{attribute 'monitoring' := 'call'}
PROPERTY PRIVATE HomeSpeedZ : LREAL
GET
HomeSpeedZ := stLocalSettings.stDynStationSettings[E_St030_Settings.eSt030_Settings_ZHomeSpeed].fValue;
END_GET
END_PROPERTY

{attribute 'monitoring' := 'call'}
PROPERTY PRIVATE IsGetCmdActive : BOOL
GET
IsGetCmdActive := stSt030IHandling.ActiveCommand.Command = E_St030_Command.eSt030_Command_OvenA_Get OR
			stSt030IHandling.ActiveCommand.Command = E_St030_Command.eSt030_Command_OvenB_Get OR
			stSt030IHandling.ActiveCommand.Command = E_St030_Command.eSt030_Command_Storage_Get;
END_GET
END_PROPERTY

{attribute 'monitoring' := 'call'}
PROPERTY PRIVATE IsGetCmdRequested : BOOL
GET
IsGetCmdRequested := stSt030IHandling.CommandRequest.Command = E_St030_Command.eSt030_Command_OvenA_Get OR
			stSt030IHandling.CommandRequest.Command = E_St030_Command.eSt030_Command_OvenB_Get OR
			stSt030IHandling.CommandRequest.Command = E_St030_Command.eSt030_Command_Storage_Get;
END_GET
END_PROPERTY

{attribute 'monitoring' := 'call'}
PROPERTY PRIVATE IsOvenCmdA : BOOL
GET
IsOvenCmdA := stSt030IHandling.ActiveCommand.Command = E_St030_Command.eSt030_Command_OvenA_Get OR
			stSt030IHandling.ActiveCommand.Command = E_St030_Command.eSt030_Command_OvenA_Put;
END_GET
END_PROPERTY

{attribute 'monitoring' := 'call'}
PROPERTY PRIVATE JogSpeedX : LREAL
GET
JogSpeedX := stLocalSettings.stDynStationSettings[E_St030_Settings.eSt030_Settings_XJogSpeed].fValue;
END_GET
END_PROPERTY

{attribute 'monitoring' := 'call'}
PROPERTY PRIVATE JogSpeedY : LREAL
GET
JogSpeedY := stLocalSettings.stDynStationSettings[E_St030_Settings.eSt030_Settings_YJogSpeed].fValue;
END_GET
END_PROPERTY

{attribute 'monitoring' := 'call'}
PROPERTY PRIVATE JogSpeedZ : LREAL
GET
JogSpeedZ := stLocalSettings.stDynStationSettings[E_St030_Settings.eSt030_Settings_ZJogSpeed].fValue;
END_GET
END_PROPERTY

METHOD PROTECTED M_CallObjects : BOOL
VAR
END_VAR
// axis + UI
fbAxisX.TorqueLimit := 600;
fbAxisX(
	bEnable := SafetyOk AND NOT fbAxisXUi.stAxisManager.bDisable AND stSt050IMould.bEnableHG,
	bEnablePos := fbAxisZ.PositionReachedWindow(PosHomeZ, 10) OR fbAxisXUi.stAxisManager.bDisableSoftLimits,
	bEnableNeg := fbAxisZ.PositionReachedWindow(PosHomeZ, 10) OR fbAxisXUi.stAxisManager.bDisableSoftLimits
);
fbAxisXUi(
	bInHome := bInHome,
	fbAxis := fbAxisX,
	fVelocity := JogSpeedX,
	diSelectedObjectIndex := stHmiManualIn.diSelectedObjectIndex,
	stHMIControlIn := stHmiManualIn.stManualAxis,
	stHMIControlOut := stHmiManualOut.stManualAxis,
	bJogP := stHmi.stIn.stSt030.bJogXP,
	bJogN := stHmi.stIn.stSt030.bJogXN,
	bEnableManual := EnableManual);

// axis CH1 + UI
fbAxisY.TorqueLimit := 600;
fbAxisY(
	bEnable := SafetyOk AND NOT fbAxisYUi.stAxisManager.bDisable AND stSt050IMould.bEnableHG,
	bEnablePos := TRUE,
	bEnableNeg := TRUE,
);
fbAxisYUi(
	bInHome := bInHome,
	fbAxis := fbAxisY,
	fVelocity := JogSpeedY,
	diSelectedObjectIndex := stHmiManualIn.diSelectedObjectIndex,
	stHMIControlIn := stHmiManualIn.stManualAxis,
	stHMIControlOut := stHmiManualOut.stManualAxis,
	bJogP := stHmi.stIn.stSt030.bJogYP,
	bJogN := stHmi.stIn.stSt030.bJogYN,
	bEnableManual := EnableManual);
	
// axis CH2 + UI
fbAxisZ.TorqueLimit := 300;
fbAxisZ(
	bEnable := SafetyOk AND NOT fbAxisZUi.stAxisManager.bDisable AND stSt050IMould.bEnableHG,
	bEnablePos := TRUE,
	bEnableNeg := TRUE,
);
fbAxisZUi(
	bInHome := bInHome,
	fbAxis := fbAxisZ,
	fVelocity := JogSpeedZ,
	diSelectedObjectIndex := stHmiManualIn.diSelectedObjectIndex,
	stHMIControlIn := stHmiManualIn.stManualAxis,
	stHMIControlOut := stHmiManualOut.stManualAxis,
	bJogP := stHmi.stIn.stSt030.bJogZP,
	bJogN := stHmi.stIn.stSt030.bJogZN,
	bEnableManual := EnableManual);
	

	
// run pallet logic
//Plant.stSt030IHandling.Pallet.Update();
END_METHOD

METHOD PRIVATE M_CheckHskRst : BOOL
VAR_INPUT
END_VAR
// chk all hand shake signals are reseted
M_CheckHskRst := FALSE;

// oven A
IF stSt010IOvenA.bResponseOpn OR stSt010IOvenA.bResponseChkIndex OR stSt010IOvenA.bResponseIsEmptySlot THEN
	sqAuto.Info.Set("warte auf Handshake reset Ofen A"); RETURN;
ELSIF stSt010IOvenA.iConfirmPosition <> -1 THEN
	sqAuto.Info.Set("warte auf Handshake Index-X reset Ofen A"); RETURN;
	
// oven B
ELSIF stSt020IOvenB.bResponseOpn OR stSt020IOvenB.bResponseChkIndex OR stSt020IOvenB.bResponseIsEmptySlot THEN
	sqAuto.Info.Set("warte auf Handshake reset Ofen B"); RETURN;
ELSIF stSt020IOvenB.iConfirmPosition <> -1 THEN
	sqAuto.Info.Set("warte auf Handshake Index-X reset Ofen B"); RETURN;
	
// storage
ELSIF stSt040IStorage.bResponseOpn OR stSt040IStorage.bResponseChkIndex OR stSt040IStorage.bResponseEmptyAtIndex THEN
	sqAuto.Info.Set("warte auf Handshake reset Storage"); RETURN;
ELSIF stSt040IStorage.iConfirmPosition <> -1 THEN
	sqAuto.Info.Set("warte auf Handshake Index reset Storage"); RETURN;
	
END_IF

M_CheckHskRst := TRUE;
END_METHOD

METHOD INTERNAL M_DynManual : BOOL
VAR_INPUT
END_VAR
IF NOT bInitManual THEN
	bInitManual := TRUE;
	MEMSET(ADR(stHmiManualOut.stObjects), 0, SIZEOF(stHmiManualOut.stObjects)); // reset
	
	M_InitDynManualUi(fbAxisXUi);
	M_InitDynManualUi(fbAxisYUi);
	M_InitDynManualUi(fbAxisZUi);
END_IF
END_METHOD

METHOD PROTECTED M_DynMonitoring : BOOL
VAR_INPUT
END_VAR
M_DynMonitoring := SUPER^.M_DynMonitoring();

// init
IF NOT bInitMonitoring THEN
	bInitMonitoring := TRUE;
	MEMSET(ADR(stLocalMonitoring), 0, SIZEOF(stLocalMonitoring)); // reset
	
	M_InitDynMonitoringItem(0, 								// monitoring index 
							"Achse X Position",				// name
							Name, 							// group (station name)
							E_DataType.eDataType_lreal, 	// data type							
							stTextListGlobal.stText_mm);	// unit	

	M_InitDynMonitoringItem(1, "Achse X Geschwindigkeit", Name, E_DataType.eDataType_lreal, stTextListGlobal.stText_mms);
	M_InitDynMonitoringItem(2, "Achse X Drehmoment", Name, E_DataType.eDataType_lreal, stTextListGlobal.stText_percent);
	
	M_InitDynMonitoringItem(4, "Achse Y Position", Name, E_DataType.eDataType_lreal, stTextListGlobal.stText_mm);
	M_InitDynMonitoringItem(5, "Achse Y Geschwindigkeit", Name, E_DataType.eDataType_lreal, stTextListGlobal.stText_mms);
	M_InitDynMonitoringItem(6, "Achse Y Drehmoment", Name, E_DataType.eDataType_lreal, stTextListGlobal.stText_percent);
	
	M_InitDynMonitoringItem(8, "Achse Z Position", Name, E_DataType.eDataType_lreal, stTextListGlobal.stText_mm);
	M_InitDynMonitoringItem(9, "Achse Z Geschwindigkeit", Name, E_DataType.eDataType_lreal, stTextListGlobal.stText_mms);
	M_InitDynMonitoringItem(10, "Achse Z Drehmoment", Name, E_DataType.eDataType_lreal, stTextListGlobal.stText_percent);
END_IF

// live value mapping 

// axis x
stLocalMonitoring.astMonitoring[0].fValue := fbAxisX.Position;
stLocalMonitoring.astMonitoring[1].fValue := fbAxisX.Velocity;
stLocalMonitoring.astMonitoring[2].fValue := fbAxisX.Torque;

// axis y
stLocalMonitoring.astMonitoring[4].fValue := fbAxisY.Position;
stLocalMonitoring.astMonitoring[5].fValue := fbAxisY.Velocity;
stLocalMonitoring.astMonitoring[6].fValue := fbAxisY.Torque;

// axis z
stLocalMonitoring.astMonitoring[8].fValue := fbAxisZ.Position;
stLocalMonitoring.astMonitoring[9].fValue := fbAxisZ.Velocity;
stLocalMonitoring.astMonitoring[10].fValue := fbAxisZ.Torque;

// hmi value mapping
//HMI.stHmi.stOut.stSt030.Pallet := stSt030IHandling.Pallet.stPallet;
END_METHOD

METHOD INTERNAL M_DynSettings : BOOL
VAR
END_VAR
// init station settings
IF NOT bInitSettings THEN
	bInitSettings := TRUE;
	stLocalSettingsBackup := stLocalSettings; // backup
	MEMSET(ADR(stLocalSettings), 0, SIZEOF(stLocalSettings)); // reset
	
	stSt030IHandling.Pallet.Config := Services.stSettings.stCarrier;
	stSt030IHandling.Pallet.InitialStatus := eTcaWorkpieceStatus.laserProcessDone;
	stSt030IHandling.Pallet.RequestStatus := eTcaWorkpieceStatus.castingProcessDone;
	stSt030IHandling.Pallet.ApplyConfig();
	
	
	M_InitDynSettingsItem(E_St030_Settings.eSt030_Settings_Station_Deaktiv,	// settings index
		TO_WSTRING(E_St030_Settings.eSt030_Settings_Station_Deaktiv),		// settings wsIndex
		Name,																// group
		stTextListGlobal.stText_DeactivateStation,							// name
		stTextListGlobal.stText_bool, E_DataType.eDataType_bool,			// unit & data type
		0, 1, 3);															// min, max & user level
    
	M_InitDynSettingsItem(E_St030_Settings.eSt030_Settings_Autohome,
		TO_WSTRING(E_St030_Settings.eSt030_Settings_Autohome),
		Name,
		stTextListGlobal.stText_AutoHome,
		stTextListGlobal.stText_bool, E_DataType.eDataType_bool,
		0, 1, 3);
		
	M_InitDynSettingsItem(E_St030_Settings.eSt030_Settings_XHomeSpeed,
		TO_WSTRING(E_St030_Settings.eSt030_Settings_XHomeSpeed),
		Name,
		F_CreateDynTextDefault("Homegeschwindigkeit Servoachse X"),
		stTextListGlobal.stText_mms, E_DataType.eDataType_lreal,
		0, 50, 3);
		
	M_InitDynSettingsItem(E_St030_Settings.eSt030_Settings_XJogSpeed,
		TO_WSTRING(E_St030_Settings.eSt030_Settings_XJogSpeed),
		Name,
		F_CreateDynTextDefault("Tippgeschwindigkeit Servoachse X"),
		stTextListGlobal.stText_mms, E_DataType.eDataType_lreal,
		0, 50, 3);
		
	M_InitDynSettingsItem(E_St030_Settings.eSt030_Settings_XWorkSpeed,
		TO_WSTRING(E_St030_Settings.eSt030_Settings_XWorkSpeed),
		Name,
		F_CreateDynTextDefault("Automatik-Geschwindigkeit Servoachse X"),
		stTextListGlobal.stText_mms, E_DataType.eDataType_lreal,
		0, 500, 3);
		
	M_InitDynSettingsItem(E_St030_Settings.eSt030_Settings_YHomeSpeed,
		TO_WSTRING(E_St030_Settings.eSt030_Settings_YHomeSpeed),
		Name,
		F_CreateDynTextDefault("Homegeschwindigkeit Servoachse Y"),
		stTextListGlobal.stText_mms, E_DataType.eDataType_lreal,
		0, 50, 3);
		
	M_InitDynSettingsItem(E_St030_Settings.eSt030_Settings_YJogSpeed,
		TO_WSTRING(E_St030_Settings.eSt030_Settings_YJogSpeed),
		Name,
		F_CreateDynTextDefault("Tippgeschwindigkeit Servoachse Y"),
		stTextListGlobal.stText_mms, E_DataType.eDataType_lreal,
		0, 50, 3);
		
	M_InitDynSettingsItem(E_St030_Settings.eSt030_Settings_YWorkSpeed,
		TO_WSTRING(E_St030_Settings.eSt030_Settings_YWorkSpeed),
		Name,
		F_CreateDynTextDefault("Automatik-Geschwindigkeit Servoachse Y"),
		stTextListGlobal.stText_mms, E_DataType.eDataType_lreal,
		0, 500, 3);
		
	M_InitDynSettingsItem(E_St030_Settings.eSt030_Settings_ZHomeSpeed,
		TO_WSTRING(E_St030_Settings.eSt030_Settings_ZHomeSpeed),
		Name,
		F_CreateDynTextDefault("Homegeschwindigkeit Servoachse Z"),
		stTextListGlobal.stText_mms, E_DataType.eDataType_lreal,
		0, 50, 3);
		
	M_InitDynSettingsItem(E_St030_Settings.eSt030_Settings_ZJogSpeed,
		TO_WSTRING(E_St030_Settings.eSt030_Settings_ZJogSpeed),
		Name,
		F_CreateDynTextDefault("Tippgeschwindigkeit Servoachse Z"),
		stTextListGlobal.stText_mms, E_DataType.eDataType_lreal,
		0, 50, 3);
		
	M_InitDynSettingsItem(E_St030_Settings.eSt030_Settings_ZWorkSpeed,
		TO_WSTRING(E_St030_Settings.eSt030_Settings_ZWorkSpeed),
		Name,
		F_CreateDynTextDefault("Automatik-Geschwindigkeit Servoachse Z"),
		stTextListGlobal.stText_mms, E_DataType.eDataType_lreal,
		0, 500, 3);
		
	M_InitDynSettingsItem(E_St030_Settings.eSt030_Settings_AxisRefPosX,	// ref pos
		TO_WSTRING(E_St030_Settings.eSt030_Settings_AxisRefPosX),
		Name,
		F_CreateDynTextDefault("Referenzposition Achse X Handling"),
		stTextListGlobal.stText_mm, E_DataType.eDataType_lreal,
		0, 1000, 6);
		
	M_InitDynSettingsItem(E_St030_Settings.eSt030_Settings_AxisRefPosY,
		TO_WSTRING(E_St030_Settings.eSt030_Settings_AxisRefPosY),
		Name,
		F_CreateDynTextDefault("Referenzposition Achse Y Handling"),
		stTextListGlobal.stText_mm, E_DataType.eDataType_lreal,
		0, 1000, 6);
		
	M_InitDynSettingsItem(E_St030_Settings.eSt030_Settings_AxisRefPosZ,
		TO_WSTRING(E_St030_Settings.eSt030_Settings_AxisRefPosZ),
		Name,
		F_CreateDynTextDefault("Referenzposition Achse Z Handling"),
		stTextListGlobal.stText_mm, E_DataType.eDataType_lreal,
		0, 1000, 6);
		
	M_InitDynSettingsItem(E_St030_Settings.eSt030_Settings_XPosHome,	// home pos
		TO_WSTRING(E_St030_Settings.eSt030_Settings_XPosHome),
		Name,
		F_CreateDynTextDefault("Homeposition Servoachse X"),
		stTextListGlobal.stText_mm, E_DataType.eDataType_lreal,
		0, 5000, 3);
	M_InitDynSettingsItem(E_St030_Settings.eSt030_Settings_YPosHome,
		TO_WSTRING(E_St030_Settings.eSt030_Settings_YPosHome),
		Name,
		F_CreateDynTextDefault("Homeposition Servoachse Y"),
		stTextListGlobal.stText_mm, E_DataType.eDataType_lreal,
		0, 3000, 3);
	M_InitDynSettingsItem(E_St030_Settings.eSt030_Settings_ZPosHome,
		TO_WSTRING(E_St030_Settings.eSt030_Settings_ZPosHome),
		Name,
		F_CreateDynTextDefault("Homeposition Servoachse Z"),
		stTextListGlobal.stText_mm, E_DataType.eDataType_lreal,
		0, 1000, 3);	

		
	// restore values
	F_RestoreSettingValues(stLocalSettings.stDynStationSettings, stLocalSettingsBackup.stDynStationSettings);
END_IF

// map current settings values to shortcuts
bStationDeaktiv := stLocalSettings.stDynStationSettings[E_St030_Settings.eSt030_Settings_Station_Deaktiv].bValue;
bAutoHome := stLocalSettings.stDynStationSettings[E_St030_Settings.eSt030_Settings_Autohome].bValue;
END_METHOD

METHOD PROTECTED M_Homing
VAR
	stHomPrm : ST_AxisHomingParameter;
END_VAR
// Homing sequence
CASE sqHome.Step OF
	
	0:	
		sqHome.Info.Set("Warte auf GRST Start");
		IF RunStep AND NOT sqHome.InHome AND bRunHoming THEN
			bBusy := TRUE;
			sqAuto.Step := 0;
			sqSearch.Step := 0;
			sqHome.StartSequence()
				  .Step := 10;
		END_IF	

	10:
		sqHome.Info.Set("Grundstellungsfahrt aktiv");
		IF P_Safety.bMachineRequestStop THEN
			sqHome.Info.Set("Anforderung Stop aktiv");
		ELSIF NOT SafetyOk THEN
			sqHome.Info.Set("Sicherheit nicht ok");
			
		ELSIF NOT fbAxisX.Operational THEN
			sqHome.Info.Set("Antrieb X nicht bereit");
		ELSIF fbAxisX.Moving THEN
			fbAxisX.Halt();
			sqHome.Info.Set("Antrieb X nicht gestoppt");
			
		ELSIF NOT fbAxisY.Operational THEN
			sqHome.Info.Set("Antrieb Y nicht bereit");
		ELSIF fbAxisY.Moving THEN
			fbAxisY.Halt();
			sqHome.Info.Set("Antrieb Y nicht gestoppt");
			
		ELSIF NOT fbAxisZ.Operational THEN
			sqHome.Info.Set("Antrieb Z nicht bereit");
		ELSIF fbAxisZ.Moving THEN
			fbAxisZ.Halt();
			sqHome.Info.Set("Antrieb Z nicht gestoppt");

		ELSIF bRunHoming THEN
			sqHome.Step := 20;
		END_IF
		
	20:	// axis Z homing
		sqHome.Info.Set("Prüfe Z-Achskalibrierung");
		IF fbAxisZ.Homed THEN
			sqHome.Step := 25;
		ELSE
			sqHome.Step := 21;
		END_IF
		
	21: 
		sqHome.Info.Set("Warte auf Referenzschalter");
		IF stIO.stIn.bRefposZ THEN
			sqHome.Step := 22;
		ELSE
			StationError.ArgSbAppendRaise('Referenzsignal Achse Z fehlt bei Referenzfahrt');
			bRunHoming := FALSE;
			sqHome.Step := 0;
		END_IF
		
	22:
		sqHome.Info.Set("Starte Z-Achskalibrierung");
		IF RunStep THEN
			stHomPrm.stOptions.SearchDirection := MC_Direction.MC_Negative_Direction;
			stHomPrm.stOptions.SyncDirection := MC_Direction.MC_Positive_Direction;
			stHomPrm.stOptions.SearchVelocity := 8;
			stHomPrm.stOptions.SyncVelocity := 4;
			stHomPrm.fPosition := HgRefPosZ;
			fbAxisZ.HomeEx(stHomPrm);
			sqHome.Step := 24;
		END_IF
		
	24:
		sqHome.Info.Set("Warte auf Z-Achskalibrierung fertig");
		fbAxisZ.bCalibrationCam := stIO.stIn.bRefposZ;
		IF fbAxisZ.Homed THEN
			sqHome.Step := 25;	
		END_IF
		
	25:
		sqHome.Info.Set("Grundstellungsfahrt aktiv Achse Z Homepos.");
		fbAxisZ.MoveAbsExVel(PosHomeZ, HomeSpeedZ);
		sqHome.Step := 26;
		
	26:
		sqHome.Info.Set("Warte auf Achse Z in Homeposition");
		IF fbAxisZ.TargetReached() THEN
			sqHome.Step := 30;	
		END_IF
		
	30:	// axis Y homing
		sqHome.Info.Set("Prüfe Y-Achskalibrierung");
		IF fbAxisY.Homed THEN
			sqHome.Step := 40;
		ELSE
			sqHome.Step := 32;
		END_IF
		
	32:
		sqHome.Info.Set("Starte Y-Achskalibrierung");
		IF RunStep THEN
			stHomPrm.stOptions.SearchDirection := MC_Direction.MC_Negative_Direction;
			stHomPrm.stOptions.SyncDirection := MC_Direction.MC_Positive_Direction;
			stHomPrm.stOptions.SearchVelocity := 8;
			stHomPrm.stOptions.SyncVelocity := 4;
			stHomPrm.fPosition := HgRefPosY;
			fbAxisY.HomeEx(stHomPrm);
			sqHome.Step := 34;
		END_IF
		
	34:
		sqHome.Info.Set("Warte auf Y-Achskalibrierung fertig");
		fbAxisY.bCalibrationCam := stIO.stIn.bRefposY;
		IF fbAxisY.Homed THEN
			sqHome.Step := 40;	
		END_IF
	
	40:	// axis X homing
		sqHome.Info.Set("Prüfe X-Achskalibrierung");
		IF fbAxisX.Homed THEN
			sqHome.Step := 50;
		ELSE
			sqHome.Step := 42;
		END_IF
		
	42:
		sqHome.Info.Set("Starte X-Achskalibrierung");
		IF RunStep THEN
			stHomPrm.stOptions.SearchDirection := MC_Direction.MC_Negative_Direction;
			stHomPrm.stOptions.SyncDirection := MC_Direction.MC_Positive_Direction;
			stHomPrm.stOptions.SearchVelocity := 8;
			stHomPrm.stOptions.SyncVelocity := 4;
			stHomPrm.fPosition := HgRefPosX;
			fbAxisX.HomeEx(stHomPrm);
			sqHome.Step := 44;
		END_IF
		
	44:
		sqHome.Info.Set("Warte auf X-Achskalibrierung fertig");
		fbAxisX.bCalibrationCam := stIO.stIn.bRefposX;
		IF fbAxisX.Homed THEN
			sqHome.Step := 50;	
		END_IF
		
	50:
		sqHome.Info.Set("Grundstellungsfahrt aktiv Achse Y Homepos.");
		fbAxisY.MoveAbsExVel(PosHomeY, HomeSpeedY);
		sqHome.Step := 55;

	55:
		sqHome.Info.Set("Warte auf Achse Y in Homeposition");
		IF fbAxisY.TargetReached() THEN
			sqHome.Step := 60;	
		END_IF
		
	60:
		sqHome.Info.Set("Grundstellungsfahrt aktiv Achse X Homepos.");
		fbAxisX.MoveAbsExVel(PosHomeX, HomeSpeedX);
		sqHome.Step := 65;
		
	65:
		sqHome.Info.Set("Warte auf Achse X in Homeposition");
		IF fbAxisX.TargetReached() AND fbAxisY.TargetReached() AND fbAxisZ.TargetReached() THEN
			M_RestActHgCmd();
			sqHome.Step := 100;	
		END_IF
		
	100:
		sqHome.Info.Set("Grundstellungsfahrt aktiv");
		sqHome.Step := 1000;

	//	homing done			
	1000:
		sqHome.Info.Set("Grundstellung erreicht");
		IF sqHome.StepTime > T#1S THEN
			bBusy:=FALSE;
			sqHome.InHome := TRUE;
			bStopped := TRUE;
			bRunHoming := FALSE;
			sqAuto.Step := 0;
			sqHome.StopSequence()
				  .Step := 0;
		END_IF
END_CASE
END_METHOD

METHOD PUBLIC M_Init : IStation
VAR_INPUT
END_VAR
VAR
	Ist : IStation;
END_VAR
// set up station
StationNb := 30;
Station := E_Station.eStation_ST030_Handling; // ID & name 1st!
Name := F_CreateDynTextEx(1, "ST030_Handling", "ST030 Handling");

Ist := SUPER^.M_Init()
			 .InitEvents(TC_Events.ST030EventClass.InfoEvent,
	  		       		 TC_Events.ST030EventClass.WarningEvent,
	  				  	 TC_Events.ST030EventClass.ErrorEvent);

// set up default IO references
M_SetReferences(IO.st030_Handling_IO);

// init components

// Axis X
fbAxisXUi.stBmk := F_CreateDynTextDefault("BMK=A03.ST30.M01-");
fbAxisXUi.stUnit := F_CreateDynTextDefault("mm");
fbAxisXUi.stAxisManager.bEnablePosSet := TRUE;
fbAxisXUi.stAxisManager.bResetCalibrationVisible := TRUE;
fbAxisXUi.stAxisManager.bSetCalibrationVisible := TRUE;
fbAxisX.AxisId := TO_INT(E_Axis.eAxis_Handling_X);
fbAxisX.Active := TRUE;
fbAxisX.Name := F_CreateDynTextEx(1, "ServoHgX", "Servoachse X");
fbAxisX.AxisType := E_AxisType.AX5xxx;
//fbAxisX.DefaultParameter := F_GetDefaultMotionParameter(eMainState_setup);
fbAxisX.SetAxisReference(NcIO.stAxis_ST030_AxisX, NcIO.stAxis_ST030_AxisX_IO.stIn, NCIO.stAxis_ST030_AxisX_IO.stOut);

// Axis CH1
fbAxisYUi.stBmk := F_CreateDynTextDefault("BMK=A03.ST30.M02-");
fbAxisYUi.stUnit := F_CreateDynTextDefault("mm");
fbAxisYUi.stAxisManager.bEnablePosSet := TRUE;
fbAxisYUi.stAxisManager.bResetCalibrationVisible := TRUE;
fbAxisYUi.stAxisManager.bSetCalibrationVisible := TRUE;
fbAxisY.AxisId := TO_INT(E_Axis.eAxis_Handling_Y);
fbAxisY.Active := TRUE;
fbAxisY.Name := F_CreateDynTextEx(1, "ServoHgY", "Servoachse Y");
fbAxisY.AxisType := E_AxisType.AX5xxx;
//fbAxisY.DefaultParameter := F_GetDefaultMotionParameter(eMainState_setup);
fbAxisY.SetAxisReference(NcIO.stAxis_ST030_AxisY, NcIO.stAxis_ST030_AxisY_IO.stIn, NCIO.stAxis_ST030_AxisY_IO.stOut);

// Axis CH2
fbAxisZUi.stBmk := F_CreateDynTextDefault("BMK=A03.ST30.M03-");
fbAxisZUi.stUnit := F_CreateDynTextDefault("mm");
fbAxisZUi.stAxisManager.bEnablePosSet := TRUE;
fbAxisZUi.stAxisManager.bResetCalibrationVisible := TRUE;
fbAxisZUi.stAxisManager.bSetCalibrationVisible := TRUE;
fbAxisZ.AxisId := TO_INT(E_Axis.eAxis_Handling_Z);
fbAxisZ.Active := TRUE;
fbAxisZ.Name := F_CreateDynTextEx(1, "ServoHgZ", "Servoachse Z");
fbAxisZ.AxisType := E_AxisType.AX5xxx;
//fbAxisZ.DefaultParameter := F_GetDefaultMotionParameter(eMainState_setup);
fbAxisZ.SetAxisReference(NcIO.stAxis_ST030_AxisZ, NcIO.stAxis_ST030_AxisZ_IO.stIn, NCIO.stAxis_ST030_AxisZ_IO.stOut);

// register station in it's module
eParent := fbModul001.M_RegisterStation(Ist);

bInitSettings	:= FALSE;
bInitMonitoring := FALSE;
bInitManual  	:= FALSE;

//aSClearText[EN] := 'Station init done.';
M_Init := Ist;
END_METHOD

METHOD PROTECTED M_Manual
VAR
END_VAR

// station must be stopped!			manual mode
IF RunCycle OR NOT bStopped THEN //(OpMode <> E_OpMode.eOpMode_manual) THEN
	RETURN;
END_IF

//IF stHmiInOut.stSt030.Command = E_HMI_PL_CMD.eHmiPlCmd_none AND_THEN 
//   stHmiInOut.stSt030.WpCmd.Command <> E_HMI_WP_CMD.eHmiWpCmd_none THEN
//	stHmiInOut.stSt030.Command := E_HMI_PL_CMD.eHmiPlCmd_performWtCmd;
//END_IF
//
//IF stHmiInOut.stSt030.Command = E_HMI_PL_CMD.eHmiPlCmd_none THEN
//	RETURN;
//END_IF
//
//stSt030IHandling.Pallet.PerformHmiCmd(stHmiInOut.stSt030);
END_METHOD

METHOD PROTECTED M_OpModeChanged : BOOL
VAR_INPUT
END_VAR
(*bBusy := FALSE;

IF (eOpMode <> eOpMode_step AND eOpMode <> eOpMode_auto) THEN
	sqAuto.Set(0);
END_IF

fbAxisX.Stop();
fbAxisY.Stop();
fbAxisZ.Stop();*)
END_METHOD

METHOD PRIVATE M_RestActHgCmd : BOOL
VAR_INPUT
END_VAR
// reset active HG command
stSt030IHandling.ActiveCommand.Command := E_St030_Command.eSt030_Command_none;
	stSt030IHandling.ActiveCommand.Position := 0;
	
stSt030IHandling.bReqestOvenA := 
stSt030IHandling.bReqestOvenA_ChkIndex := 
stSt030IHandling.bReqestOvenB := 
stSt030IHandling.bReqestOvenB_ChkIndex := 
stSt030IHandling.bReqestStorage :=
stSt030IHandling.bReqestStorage_ChkIndex := FALSE;
END_METHOD

METHOD PUBLIC M_Run : BOOL
VAR_INPUT
END_VAR
// check refs valid
IF NOT __ISVALIDREF(stIO) THEN
	RETURN;
END_IF

M_RUN := SUPER^.M_Run();

M_DynSettings();
M_DynManual();
M_DynMonitoring();
END_METHOD

METHOD PROTECTED M_Sequence
VAR
	wsCurJob : WSTRING; 
END_VAR
// signal mapping (e.g.: enable)
stSt030IHandling.bEnable := (sqAuto.Step >= 100 AND sqAuto.Step <= 500) OR
									 bStationDeaktiv;
stSt030IHandling.bEnableOvenAxis := fbAxisZ.PositionReachedWindow(PosHomeZ, 30);
									 
wsCurJob := TO_WSTRING(stSt030IHandling.ActiveCommand.Command);

// automatic sequence
CASE sqAuto.Step OF
		
	0:	sqAuto.Info.Set("Warte auf Auto Start");
		IF RunCycle AND RunStep THEN
			//sqAuto.Info.Set("Warte auf GRST");
			//IF sqHome.InHome AND bInHome THEN
				sqHome.InHome := FALSE;
				sqAuto.Step := 5;
			//ELSE
			//	StationError.ArgSbAppendWsRaise(stTextlistGlobal.stText_station_not_in_hp);
			//END_IF
		END_IF
		
	5:	IF bStationDeaktiv THEN
			sqAuto.Info.Set("Station deaktiv");
		ELSE
			sqAuto.Step := 10;
		END_IF
		
	10:	sqAuto.Info.Set("Prüfe Startbedingungen");
		IF NOT (fbAxisX.Operational AND fbAxisX.Homed) THEN
			StationError.ArgSbAppendRaise('Bereitsignal Achse X fehlt');
		ELSIF NOT (fbAxisY.Operational AND fbAxisY.Homed) THEN
			StationError.ArgSbAppendRaise('Bereitsignal Achse Y fehlt');
		ELSIF NOT (fbAxisZ.Operational AND fbAxisZ.Homed) THEN
			StationError.ArgSbAppendRaise('Bereitsignal Achse Z fehlt');
		ELSE
			CycleStart();
			sqAuto.SetStep(15);
		END_IF
		
	15: sqAuto.Info.Set("Prüfe Job-Anforderung");
		IF stSt030IHandling.CommandRequest.Command = E_St030_Command.eSt030_Command_none THEN
			sqAuto.SetStep(20);	// home
		ELSE
			sqAuto.SetStep(100);
		END_IF
		
	// hg to travel/home position
	20: sqAuto.Info.Set("Grundstellungsfahrt aktiv Achse Z Homepos.");
		fbAxisZ.MoveAbsExVel(PosHomeZ, WorkSpeedZ);
		sqAuto.Step := 25;
	
	25: sqAuto.Info.Set("Warte auf Achse Z in Homeposition");
		IF fbAxisZ.TargetReached() THEN
			sqAuto.SetStep(30);	
		END_IF
		
	30: sqAuto.Info.Set("Grundstellungsfahrt aktiv Achse Y Homepos.");
		fbAxisY.MoveAbsExVel(PosHomeY, WorkSpeedY);
		sqAuto.Step := 35;

	35: sqAuto.Info.Set("Warte auf Achse Y in Homeposition");
		IF fbAxisY.TargetReached() THEN
			sqAuto.Step := 100;
		END_IF
		
	// work
	100: sqAuto.Info.Set("Automatik, warte auf Job");
		M_RestActHgCmd();
		IF NOT RunCycle THEN sqAuto.Step := 900; RETURN; END_IF
		IF NOT M_CheckHskRst() THEN RETURN; END_IF
		
		IF IsGetCmdRequested AND stSt030IHandling.Pallet.CarrierPresent THEN
			StationWarning.ArgSbAppendRaise('Palette bereits auf HG bei Abhol-Auftrag');
			RETURN;
		END_IF
		
		stSt030IHandling.ActiveCommand := stSt030IHandling.CommandRequest;
		IF stSt030IHandling.ActiveCommand.Command <> E_St030_Command.eSt030_Command_none THEN
			sqAuto.Step := 110;
		END_IF
		
	// hg switch job
	110: sqAuto.Info.Set("Automatik, Job: ")
					.Append(TO_WSTRING(stSt030IHandling.ActiveCommand.Command));
		CASE stSt030IHandling.ActiveCommand.Command OF
			E_St030_Command.eSt030_Command_OvenA_Get,
			E_St030_Command.eSt030_Command_OvenA_Put,			
			E_St030_Command.eSt030_Command_OvenB_Get,
			E_St030_Command.eSt030_Command_OvenB_Put: sqAuto.SetStep(300);
			
			E_St030_Command.eSt030_Command_Storage_Get,
			E_St030_Command.eSt030_Command_Storage_Put: sqAuto.SetStep(500);
		END_CASE
		
	// get/put oven A/B
	300: sqAuto.Info.Set("Job: ")
					.Append(wsCurJob).Append(", ")
					.Append("Achse X positionieren");
		fbAxisX.MoveAbsExVel(PosWorkOvenX, WorkSpeedX);
		sqAuto.Step := 305;
		
	305: sqAuto.Info.Set("Job: ")
					.Append(wsCurJob).Append(", ")
					.Append("warte auf Achse X in Pos.");
		IF fbAxisX.TargetReached() THEN
			sqAuto.SetStep(310);
		END_IF
					
	310: sqAuto.Info.Set("Job: ")
					.Append(wsCurJob).Append(", ")
					.Append("Achse Y positionieren");
					
		fbAxisY.MoveAbsExVel(SEL(IsGetCmdActive, PosWorkOvenY_OffsUp, PosWorkOvenY_OffsDn),
							 WorkSpeedY);
		sqAuto.Step := 315;
		
	315: sqAuto.Info.Set("Job: ")
					.Append(wsCurJob).Append(", ")
					.Append("warte auf Achse Y in Pos.");
		IF fbAxisY.TargetReached() THEN
			sqAuto.SetStep(320);
		END_IF
		
	320: sqAuto.Info.Set("Job: ")
					.Append(wsCurJob).Append(", ")
					.Append("Achse Z positionieren");
		fbAxisZ.MoveAbsExVel(PosHomeZ, WorkSpeedZ);
		sqAuto.Step := 325;
		
	325: sqAuto.Info.Set("Job: ")
					.Append(wsCurJob).Append(", ")
					.Append("warte auf Achse Z in Pos.");
		IF fbAxisZ.TargetReached() THEN
			sqAuto.Step := 330;
		END_IF
					
	330: sqAuto.Info.Set("Job: ")
					.Append(wsCurJob).Append(", ")
					.Append("prüfe Status: ");
		IF IsOvenCmdA THEN
			sqAuto.Info.Append("Index, ");
			stSt030IHandling.bReqestOvenA_ChkIndex := TRUE;
			IF NOT stSt010IOvenA.bResponseChkIndex THEN RETURN; END_IF
			sqAuto.Info.Append("Position, ");
			IF stSt010IOvenA.iConfirmPosition <> stSt030IHandling.ActiveCommand.Position THEN RETURN; END_IF
			sqAuto.Info.Append("Pallet");
			IF stSt030IHandling.ActiveCommand.Command = E_St030_Command.eSt030_Command_OvenA_Put AND NOT stSt010IOvenA.bResponseIsEmptySlot THEN 
				StationError.ArgSbAppendRaise('Ablage auf belegte Position!');
				RETURN;
			END_IF
		ELSE
			sqAuto.Info.Append("Index, ");
			stSt030IHandling.bReqestOvenB_ChkIndex := TRUE;
			IF NOT stSt020IOvenB.bResponseChkIndex THEN RETURN; END_IF
			sqAuto.Info.Append("Position, ");
			IF stSt020IOvenB.iConfirmPosition <> stSt030IHandling.ActiveCommand.Position THEN RETURN; END_IF
			sqAuto.Info.Append("Pallet");
			IF stSt030IHandling.ActiveCommand.Command = E_St030_Command.eSt030_Command_OvenB_Put AND NOT stSt020IOvenB.bResponseIsEmptySlot THEN
	 			StationError.ArgSbAppendRaise('Ablage auf belegte Position!');
				RETURN;
			END_IF
		END_IF
		sqAuto.Step := 340;
		
	340: sqAuto.Info.Set("Job: ")
					.Append(wsCurJob).Append(", ")
					.Append("warte auf Segment offen.");
		IF IsOvenCmdA THEN
			stSt030IHandling.bReqestOvenA := TRUE;
			IF NOT stSt010IOvenA.bResponseOpn THEN RETURN; END_IF
		ELSE
			stSt030IHandling.bReqestOvenB := TRUE;
			IF NOT stSt020IOvenB.bResponseOpn THEN RETURN; END_IF
		END_IF
		sqAuto.SetStep(350);
		
//ToDo: chk hier ev. X-Suchfahrt?
	345: sqAuto.Info.Set(sqSearch.Info.ToWString());
		IF sqAuto.Init THEN sqSearch.Step := 10; END_IF
		IF sqSearch.Step = 0 THEN
			sqAuto.SetStep(350);
		END_IF
		
	350: sqAuto.Info.Set("Job: ")
					.Append(wsCurJob).Append(", ")
					.Append("Achse Z positionieren");
		fbAxisZ.MoveAbsExVel(PosWorkOvenZ, WorkSpeedZ);
		sqAuto.Step := 355;
		
	355: sqAuto.Info.Set("Job: ")
					.Append(wsCurJob).Append(", ")
					.Append("warte auf Achse Z in Pos.");
		IF fbAxisZ.TargetReached() THEN
			sqAuto.SetStep(360);
		END_IF
		
	360: sqAuto.Info.Set("Job: ")
					.Append(wsCurJob).Append(", ")
					.Append("Achse Y positionieren");
					
		fbAxisY.MoveAbsExVel(SEL(IsGetCmdActive, PosWorkOvenY_OffsDn, PosWorkOvenY_OffsUp),
							 WorkSpeedY);
		sqAuto.Step := 365;
		
	365: sqAuto.Info.Set("Job: ")
					.Append(wsCurJob).Append(", ")
					.Append("warte auf Achse Y in Pos.");
		IF fbAxisY.TargetReached() THEN
			sqAuto.SetStep(SEL(IsGetCmdActive, 367, 366));
		END_IF
		
	366: sqAuto.Info.Set("Übernehme Teiledaten Ofen -> HG");
		IF IsOvenCmdA THEN
			stSt030IHandling.Pallet.SetCarrier(
				stSt010IOvenA.Trolley.GetCarrierAt(stSt010IOvenA.iConfirmPosition));
				stSt030IHandling.Source := E_Station.eStation_ST010_OvenA;
				
			//TODO: Daten am Handling löschen
			stSt010IOvenA.Trolley.RemoveCarrierAt(stSt010IOvenA.iConfirmPosition);
				
		ELSE
			stSt030IHandling.Pallet.SetCarrier(
				stSt020IOvenB.Trolley.GetCarrierAt(stSt020IOvenB.iConfirmPosition));
				stSt030IHandling.Source := E_Station.eStation_ST020_OvenB;
					
			//TODO: Daten am Handling löschen		
			stSt020IOvenB.Trolley.RemoveCarrierAt(stSt010IOvenA.iConfirmPosition);
		END_IF	
		sqAuto.Step := 368;
		
	367: sqAuto.Info.Set("Übernehme Teiledaten HG -> Ofen");
		IF IsOvenCmdA THEN
			stSt010IOvenA.Trolley.SetCarrierAt(stSt010IOvenA.iConfirmPosition,
											  stSt030IHandling.Pallet.Data);
		ELSE
			stSt020IOvenB.Trolley.SetCarrierAt(stSt020IOvenB.iConfirmPosition,
											  stSt030IHandling.Pallet.Data);
		END_IF
		//TODO: Daten am Handling löschen
		stSt030IHandling.Pallet.RemoveCarrier();
		stSt030IHandling.Source := E_Station.eStation_none;
		sqAuto.Step := 368;
		
	368: sqAuto.Info.Set("Übernehme Teiledaten HG -> Ofen");
		sqAuto.SetStep(370);
		
	370: sqAuto.Info.Set("Job: ")
					.Append(wsCurJob).Append(", ")
					.Append("warte auf Achse Z in Pos.");
		fbAxisZ.MoveAbsExVel(PosHomeZ, WorkSpeedZ);
		sqAuto.Step := 375;
	
	375: sqAuto.Info.Set("Job: ")
					.Append(wsCurJob).Append(", ")
					.Append("warte auf Achse Z in Pos.");
		IF fbAxisZ.TargetReached() THEN
			sqAuto.SetStep(380);
		ELSIF fbAxisZ.TargetWindowReached(2) THEN
			stSt030IHandling.bReqestOvenA := 
			stSt030IHandling.bReqestOvenB := FALSE; // cls segment as soon as possible
		END_IF
		
	380: sqAuto.Info.Set("Job: ")
					.Append(wsCurJob).Append(", ")
					.Append("warte auf Segment geschlossen.");
		IF IsOvenCmdA THEN
			stSt030IHandling.bReqestOvenA := FALSE;
			IF stSt010IOvenA.bResponseOpn THEN RETURN; END_IF
		ELSE
			stSt030IHandling.bReqestOvenB := FALSE;
			IF stSt020IOvenB.bResponseOpn THEN RETURN; END_IF
		END_IF
		sqAuto.Step := 800; // step done
			  
		
	// get/put storage
	500: sqAuto.Info.Set("Job: ")
					.Append(wsCurJob).Append(", ")
					.Append("Achse X positionieren");
		fbAxisX.MoveAbsExVel(PosWorkStorageX, WorkSpeedX);
		sqAuto.Step := 505;
		
	505: sqAuto.Info.Set("Job: ")
					.Append(wsCurJob).Append(", ")
					.Append("warte auf Achse X in Pos.");
		IF fbAxisX.TargetReached() THEN
			sqAuto.SetStep(510);
		END_IF
					
	510: sqAuto.Info.Set("Job: ")
					.Append(wsCurJob).Append(", ")
					.Append("Achse Y positionieren");
					
		fbAxisY.MoveAbsExVel(SEL(IsGetCmdActive, PosWorkStorageY_OffsUp, PosWorkStorageY_OffsDn),
							 WorkSpeedY);
		sqAuto.Step := 515;
		
	515: sqAuto.Info.Set("Job: ")
					.Append(wsCurJob).Append(", ")
					.Append("warte auf Achse Y in Pos.");
		IF fbAxisY.TargetReached() THEN
			sqAuto.SetStep(520);
		END_IF
		
	520: sqAuto.Info.Set("Job: ")
					.Append(wsCurJob).Append(", ")
					.Append("Achse Z positionieren");
		fbAxisZ.MoveAbsExVel(PosHomeZ, WorkSpeedZ);
		sqAuto.Step := 525;
		
	525: sqAuto.Info.Set("Job: ")
					.Append(wsCurJob).Append(", ")
					.Append("warte auf Achse Z in Pos.");
		IF fbAxisZ.TargetReached() THEN
			sqAuto.Step := 530;
		END_IF
		
	530: sqAuto.Info.Set("Job: ")
					.Append(wsCurJob).Append(", ")
					.Append("prüfe Status: Index, ");
		stSt030IHandling.bReqestStorage_ChkIndex := TRUE;
		IF NOT stSt040IStorage.bResponseChkIndex THEN RETURN; END_IF
		sqAuto.Info.Append("Position, ");
		IF stSt040IStorage.iConfirmPosition <> stSt030IHandling.ActiveCommand.Position THEN RETURN; END_IF
		sqAuto.Info.Append("Pallet");
		IF stSt040IStorage.bResponseEmptyAtIndex OR stSt030IHandling.ActiveCommand.Command = E_St030_Command.eSt030_Command_Storage_Get THEN 
			sqAuto.Step := 540;
		END_IF		
		
	540: sqAuto.Info.Set("Job: ")
					.Append(wsCurJob).Append(", ")
					.Append("warte auf Storage offen.");
		stSt030IHandling.bReqestStorage := TRUE;
		IF NOT stSt040IStorage.bResponseOpn THEN RETURN; END_IF
		sqAuto.SetStep(550);
		
	550: sqAuto.Info.Set("Job: ")
					.Append(wsCurJob).Append(", ")
					.Append("Achse Z positionieren");
		fbAxisZ.MoveAbsExVel(PosWorkStorageZ, WorkSpeedZ);
		sqAuto.Step := 555;
		
	555: sqAuto.Info.Set("Job: ")
					.Append(wsCurJob).Append(", ")
					.Append("warte auf Achse Z in Pos.");
		IF fbAxisZ.TargetReached() THEN
			sqAuto.SetStep(560);
		END_IF
		
	560: sqAuto.Info.Set("Job: ")
					.Append(wsCurJob).Append(", ")
					.Append("Achse Y positionieren");
					
		fbAxisY.MoveAbsExVel(SEL(IsGetCmdActive, PosWorkStorageY_OffsDn, PosWorkStorageY_OffsUp),
							 WorkSpeedY);
		sqAuto.Step := 565;
		
	565: sqAuto.Info.Set("Job: ")
					.Append(wsCurJob).Append(", ")
					.Append("warte auf Achse Y in Pos.");
		IF fbAxisY.TargetReached() THEN
			sqAuto.SetStep(SEL(IsGetCmdActive, 567, 566));
		END_IF
		
	566: sqAuto.Info.Set("Übernehme Teiledaten Storage -> HG");
		IF stSt030IHandling.ActiveCommand.Position = 1 THEN
			stSt030IHandling.Pallet.SetCarrier(
				stSt040IStorage.Pallet1.Data);
			stSt030IHandling.Source := stSt040IStorage.Source1;
			//TODO Storagedaten löschen	
			stSt040IStorage.Pallet1.RemoveCarrier();
			stSt040IStorage.Source1 := E_Station.eStation_none;
		
		ELSIF stSt030IHandling.ActiveCommand.Position = 2 THEN
			stSt030IHandling.Pallet.SetCarrier(
				stSt040IStorage.Pallet2.Data);
			stSt030IHandling.Source := stSt040IStorage.Source2;
			//TODO Storagedaten löschen	
			stSt040IStorage.Pallet2.RemoveCarrier();
			stSt040IStorage.Source2 := E_Station.eStation_none;
		END_IF
		
		sqAuto.Step := 568;
		
	567: sqAuto.Info.Set("Übernehme Teiledaten HG -> Storage");
		IF  stSt030IHandling.ActiveCommand.Position = 1 THEN
			stSt040IStorage.Pallet1.SetCarrier(
				stSt030IHandling.Pallet.Data);
			stSt040IStorage.Source1 := stSt030IHandling.Source;
		ELSIF stSt030IHandling.ActiveCommand.Position = 2 THEN
			stSt040IStorage.Pallet2.SetCarrier(
				stSt030IHandling.Pallet.Data);
			stSt040IStorage.Source2 := stSt030IHandling.Source; 
		END_IF
		sqAuto.Step := 568;
		
	568: sqAuto.Info.Set("Übernehme Teiledaten");
		sqAuto.SetStep(570);
		
	570: sqAuto.Info.Set("Job: ")
					.Append(wsCurJob).Append(", ")
					.Append("warte auf Achse Z in Pos.");
		fbAxisZ.MoveAbsExVel(PosHomeZ, WorkSpeedZ);
		sqAuto.Step := 575;
	
	575: sqAuto.Info.Set("Job: ")
					.Append(wsCurJob).Append(", ")
					.Append("warte auf Achse Z in Pos.");
		IF fbAxisZ.TargetReached() THEN
			sqAuto.SetStep(580);
		ELSIF fbAxisZ.TargetWindowReached(2) THEN
			stSt030IHandling.bReqestStorage := FALSE; // cls stoarge as soon as possible
		END_IF
		
	580: sqAuto.Info.Set("Job: ")
					.Append(wsCurJob).Append(", ")
					.Append("warte auf Storage geschlossen.");
		stSt030IHandling.bReqestStorage := FALSE;
		IF stSt040IStorage.bResponseOpn THEN RETURN; END_IF
		sqAuto.Step := 800; // step done
		
	// job done
	800: sqAuto.Info.Set("Job fertig, warte Handshake reset");
		IF stSt030IHandling.CommandRequest.Command = E_St030_Command.eSt030_Command_none OR
		   stSt030IHandling.CommandRequest.Command <> stSt030IHandling.ActiveCommand.Command THEN
			sqAuto.SetStep(900);
		END_IF
		
	// rdy	
	900: sqAuto.Info.Set("Zyklus beendet");
		CycleEnd();
		sqAuto.Step := 0;

	// error
	1000: sqAuto.Info.Set("Error");
		bStopped := TRUE;
		sqHome.InHome := FALSE;
		bRunHoming := FALSE;

END_CASE
END_METHOD

METHOD INTERNAL M_SequenceSearch : ST_Text
VAR_INST
	rfTrigS1,
	rfTrigS2 	: FB_RtrigFtrig;
	fPos 		: LREAL;
END_VAR
IF sqSearch.Step < 10 THEN RETURN; END_IF
rfTrigS1(bIn := MeasurementA >= fThreshMesMin AND MeasurementA <= fThreshMesMax);
rfTrigS2(bIn := MeasurementB >= fThreshMesMin AND MeasurementB <= fThreshMesMax);
sqSearch.EnableStep := RunStep;

// search sequence
CASE sqSearch.Step OF
		
	0:	sqSearch.Info.Set("Warte auf Start Suche");
		
	10:	sqSearch.Info.Set("Start Suche, Backup HG-Position");
		fPosSearchCorr := 0;
		eEmptyChk := E_St030_EmptySlotChk.eSt030_EmptySlotChk_none;
		HgPosBackup.x := fbAxisX.Position;
		HgPosBackup.y := fbAxisY.Position;
		HgPosBackup.z := fbAxisZ.Position;
		sqSearch.SetStep(20);
		
	// hg to start search position
	20: sqSearch.Info.Set("Suche aktiv Achse Z");
		fbAxisZ.MoveAbsExVel(PosHomeZ, WorkSpeedZ);
		sqSearch.Step := 25;
	
	25: sqSearch.Info.Set("Warte auf Achse Z in Such-Pos. 1");
		IF fbAxisZ.TargetReached() THEN
			sqSearch.SetStep(30);	
		END_IF
		
	30: sqSearch.Info.Set("Suche aktiv Achse X");
		fbAxisX.MoveAbsExVel(PosWorkOvenX - 25, WorkSpeedX);
		sqSearch.Step := 35;
		
	35: sqSearch.Info.Set("Warte auf Achse X in Such-Pos. 1");
		IF fbAxisX.TargetReached() THEN
			sqSearch.SetStep(40);
		END_IF	
		
	40: sqSearch.Info.Set("Suche aktiv Achse Y");
		fbAxisY.MoveAbsExVel(PosWorkOvenY_OffsDn, WorkSpeedY);
		sqSearch.Step := 45;

	45: sqSearch.Info.Set("Warte auf Achse Y in Such-Pos. 1");
		IF fbAxisY.TargetReached() THEN
			sqSearch.SetStep(50);
		END_IF
		
	// chk sensor start condition, start search..
	50: sqSearch.Info.Set("Check Startbedingungen Suchfahrt 1");
		IF rfTrigS1.bIn THEN
			StationError.ArgSbAppendRaise('Signal Sensor S1 steht noch an');
		ELSIF rfTrigS2.bIn THEN
			StationError.ArgSbAppendRaise('Signal Sensor S2 steht noch an');
		ELSE
			fbAxisX.MoveAbsExVel(PosWorkOvenX, HomeSpeedX);
			MEMSET(ADR(SearchTrig), 0, SIZEOF(SearchTrig));
			sqSearch.Step := 60;
		END_IF
	
	60: sqSearch.Info.Set("Suchfahrt 1 aktiv (Achse X)");
		IF rfTrigS1.bRq THEN 
			SearchTrig[0, 0].X := fbAxisX.Position;
			SearchTrig[0, 0].Z := MeasurementA;
		END_IF
		IF rfTrigS2.bRq THEN 
			SearchTrig[1, 0].X := fbAxisX.Position;
			SearchTrig[1, 0].Z := MeasurementB;
		END_IF
		IF SearchTrig[0, 0].X <> 0 AND SearchTrig[1, 0].X <> 0 THEN
			sqSearch.SetStep(80);
		ELSIF sqSearch.SeqTime > T#10S THEN
			StationError.ArgSbAppendRaise('Timeout Suchfahrt 1');
		END_IF
		
	80: sqSearch.Info.Set("Check Startbedingungen Suchfahrt 2");
		IF NOT rfTrigS1.bIn THEN
			StationError.ArgSbAppendRaise('Signal Sensor S1 fehlt');
		ELSIF NOT rfTrigS2.bIn THEN
			StationError.ArgSbAppendRaise('Signal Sensor S2 fehlt');
		ELSE
			fbAxisX.MoveAbsExVel(PosWorkOvenX + 25, HomeSpeedX);
			sqSearch.Step := 90;
		END_IF
	
	90: sqSearch.Info.Set("Suchfahrt 2 aktiv (Achse X)");
		IF rfTrigS1.bFq THEN 
			SearchTrig[0, 1].X := fbAxisX.Position;
			SearchTrig[0, 1].Z := MeasurementA;
		END_IF
		IF rfTrigS2.bFq THEN 
			SearchTrig[1, 1].X := fbAxisX.Position;
			SearchTrig[1, 1].Z := MeasurementB;
		END_IF
		IF SearchTrig[0, 1].X <> 0 AND SearchTrig[1, 1].X <> 0 THEN
			sqSearch.Step := 300;
		ELSIF sqSearch.SeqTime > T#100S THEN
			StationError.ArgSbAppendRaise('Timeout Suchfahrt 2');
		END_IF
		
	100: sqSearch.Info.Set("Auswertung Suchfahrt..");
		//IF ABS(SearchTrig[0, 0] - SearchTrig[0, 1]) > 2 THEN
		//	INotiHdl.M_SetNotiDefaultErr(stTextlistGlobal.stText_NG_Stations, Name, F_CreateDynTextDefault("Trigger-Signale Sensor S1 unplausibel"), stEmptyText);
		//ELSIF ABS(SearchTrig[1, 0] - SearchTrig[1, 1]) > 2 THEN
		//	INotiHdl.M_SetNotiDefaultErr(stTextlistGlobal.stText_NG_Stations, Name, F_CreateDynTextDefault("Trigger-Signale Sensor S2 unplausibel"), stEmptyText);
		//ELSE
			//fPosSearchCorr := ((SearchTrig[0, 0] - SearchTrig[0, 1]) + (SearchTrig[1, 0] - SearchTrig[1, 1]))/2;
			sqSearch.SetStep(200);
		//END_IF
	
	// hg to chk empty slot position
	200: sqSearch.Info.Set("Suche aktiv Achse X");
		fbAxisX.MoveAbsExVel(PosWorkOvenX + 50, WorkSpeedX);
		fbAxisY.MoveAbsExVel(PosWorkOvenY - 25, WorkSpeedY); //ToDo: chk pos!
		sqSearch.Step := 205;
		
	205: sqSearch.Info.Set("Warte auf Achse X in Slot-Check-Pos.");
		IF NOT fbAxisX.TargetReached() THEN RETURN; END_IF
		sqSearch.Info.Set("Warte auf Achse Y in Slot-Check-Pos.");
		IF NOT fbAxisY.TargetReached() THEN RETURN; END_IF
		sqSearch.Step := 210;
		
	210: sqSearch.Info.Set("Suche aktiv Achse Y");
		eEmptyChk := SEL(rfTrigS1.bIn, E_St030_EmptySlotChk.eSt030_EmptySlotChk_Empty, E_St030_EmptySlotChk.eSt030_EmptySlotChk_NotEmpty);
		sqSearch.SetStep(300);		
	
	// hg to backup position
	300: sqSearch.Info.Set("Wiederherstellung HG aktiv Achse Z");
		fbAxisZ.MoveAbsExVel(HgPosBackup.z, WorkSpeedZ);
		sqSearch.Step := 305;
	
	305: sqSearch.Info.Set("Warte auf Achse Z in Backupposition");
		IF fbAxisZ.TargetReached() THEN
			sqSearch.SetStep(310);	
		END_IF
		
	310: sqSearch.Info.Set("Wiederherstellung aktiv Achse Y");
		fbAxisY.MoveAbsExVel(HgPosBackup.y, WorkSpeedY);
		sqSearch.Step := 315;

	315: sqSearch.Info.Set("Warte auf Achse Y in Backupposition");
		IF fbAxisY.TargetReached() THEN
			sqSearch.SetStep(320);	
		END_IF
		
	320: sqSearch.Info.Set("Wiederherstellung aktiv Achse X");
		fbAxisX.MoveAbsExVel(HgPosBackup.x, WorkSpeedX);
		sqSearch.Step := 325;
		
	325: sqSearch.Info.Set("Warte auf Achse X in Backupposition");
		IF fbAxisX.TargetReached() AND fbAxisY.TargetReached() AND fbAxisZ.TargetReached() THEN
			sqSearch.Step := 0;
		END_IF
	
END_CASE
END_METHOD

METHOD INTERNAL M_SetReferences : BOOL
VAR_IN_OUT
	stIoRef : ST_St030_IO;
END_VAR
stIO REF= stIoRef;
M_SetReferences := TRUE;
END_METHOD

METHOD PROTECTED M_Supervision : BOOL
VAR
END_VAR
// chk stopped
IF NOT bRunCycle OR P_Safety.bMachineRequestStop THEN
	IF P_Safety.bMachineRequestStop THEN
		fbAxisX.Stop();
		fbAxisY.Stop();
		fbAxisZ.Stop();
	END_IF
	IF sqAuto.StepTime > T#20S THEN
		bStopped := TRUE;
	END_IF
END_IF

// axis x
IF fbAxisX.bError THEN
	ReactToComponentError(fbAxisXUi, E_EventReaction.Stop);

// y
ELSIF fbAxisY.bError THEN
	ReactToComponentError(fbAxisYUi, E_EventReaction.Stop);
	
// z
ELSIF fbAxisZ.bError THEN
	ReactToComponentError(fbAxisZUi, E_EventReaction.Stop);
	
END_IF
END_METHOD

{attribute 'monitoring' := 'call'}
PROPERTY INTERNAL MeasurementA : LREAL
GET
MeasurementA := TO_LREAL(stIO.stIn.fMeasurementA)/1E3;
END_GET
END_PROPERTY

{attribute 'monitoring' := 'call'}
PROPERTY INTERNAL MeasurementB : LREAL
GET
MeasurementB := TO_LREAL(stIO.stIn.fMeasurementB)/1E3;
END_GET
END_PROPERTY

{attribute 'monitoring' := 'call'}
PROPERTY PRIVATE PosHomeX : LREAL
GET
PosHomeX := stLocalSettings.stDynStationSettings[E_St030_Settings.eSt030_Settings_XPosHome].fValue;
END_GET
END_PROPERTY

{attribute 'monitoring' := 'call'}
PROPERTY PRIVATE PosHomeY : LREAL
GET
PosHomeY := stLocalSettings.stDynStationSettings[E_St030_Settings.eSt030_Settings_YPosHome].fValue;
END_GET
END_PROPERTY

{attribute 'monitoring' := 'call'}
PROPERTY PRIVATE PosHomeZ : LREAL
GET
PosHomeZ := stLocalSettings.stDynStationSettings[E_St030_Settings.eSt030_Settings_ZPosHome].fValue;
END_GET
END_PROPERTY

{attribute 'monitoring' := 'call'}
PROPERTY PRIVATE PosWorkOvenX : LREAL
GET
VAR
	iOven 		: INT;
	fDeltaX, fDeltaY,
	fRp1, fRp2,
	fApprox,
	fDevision 	: LREAL;
END_VAR
// set oven (A/B --> 1/2)
iOven := 	SEL(stSt030IHandling.ActiveCommand.Command = E_St030_Command.eSt030_Command_OvenA_Get OR
				stSt030IHandling.ActiveCommand.Command = E_St030_Command.eSt030_Command_OvenA_Put, 2, 1);
				
// calc x-approximation
fRp1 := GetPosOvRp(iOven, 1, 'Y');
fRp2 := GetPosOvRp(iOven, 2, 'Y');
fDeltaY := fRp2 - fRp1;


fRp1 := GetPosOvRp(iOven, 1, 'X');
fRp2 := GetPosOvRp(iOven, 2, 'X');
fDeltaX := fRp2 - fRp1;	

IF ABS(fDeltaY) > fEpsilon THEN
	fApprox := fDeltaX/fDeltaY * (PosWorkOvenY - fRp1);
END_IF

// ..IndexX = 1 => - Teilung, ..IndexX = 2 => + Teilung
fDevision := P_Plant.TrolleyRackDivision * SEL(stSt030IHandling.ActiveCommand.Position = 1, -0.5, 0.5);

PosWorkOvenX := SEL(iOven = 2, Plant.fbSt010OvenA.OvenMiddlePointX, Plant.fbSt020OvenB.OvenMiddlePointX) +
				fDevision + fApprox;
END_GET
END_PROPERTY

{attribute 'monitoring' := 'call'}
PROPERTY PRIVATE PosWorkOvenY : LREAL
GET
VAR
	iOven 		: INT;
END_VAR
// set oven (A/B --> 1/2)
iOven := 	SEL(stSt030IHandling.ActiveCommand.Command = E_St030_Command.eSt030_Command_OvenA_Get OR
				stSt030IHandling.ActiveCommand.Command = E_St030_Command.eSt030_Command_OvenA_Put, 2, 1);

PosWorkOvenY := (P_Plant.TrolleyCarrierDistance * stSt030IHandling.ActiveCommand.Position) + 
					P_Plant.TrolleyRackOriginY + 
					SEL(iOven = 2, Plant.fbSt010OvenA.OvenOffsetY, Plant.fbSt020OvenB.OvenOffsetY);
END_GET
END_PROPERTY

{attribute 'monitoring' := 'call'}
PROPERTY PRIVATE PosWorkOvenY_OffsDn : LREAL
GET
PosWorkOvenY_OffsDn := PosWorkOvenY - 15;// P_Plant.TrolleyOffsetDnY; //15
END_GET
END_PROPERTY

{attribute 'monitoring' := 'call'}
PROPERTY PRIVATE PosWorkOvenY_OffsUp : LREAL
GET
PosWorkOvenY_OffsUp := PosWorkOvenY + 20;//P_Plant.TrolleyOffsetUpY; //20
END_GET
END_PROPERTY

{attribute 'monitoring' := 'call'}
PROPERTY PRIVATE PosWorkOvenZ : LREAL
GET
VAR
	iOven 		: INT;
	fDeltaZ, fDeltaY,
	fRp1, fRp2,
	fApprox		: LREAL;
END_VAR
// set oven (A/B --> 1/2)
iOven := 	SEL(stSt030IHandling.ActiveCommand.Command = E_St030_Command.eSt030_Command_OvenA_Get OR
				stSt030IHandling.ActiveCommand.Command = E_St030_Command.eSt030_Command_OvenA_Put, 2, 1);
				
// calc x-approximation
fRp1 := GetPosOvRp(iOven, 1, 'Y');
fRp2 := GetPosOvRp(iOven, 2, 'Y');
fDeltaY := fRp2 - fRp1;

fRp1 := GetPosOvRp(iOven, 1, 'Z');
fRp2 := GetPosOvRp(iOven, 2, 'Z');
fDeltaZ := fRp2 - fRp1;

IF ABS(fDeltaY) > fEpsilon THEN
	fApprox := fDeltaZ/fDeltaY * (PosWorkOvenY - fRp1);
END_IF

PosWorkOvenZ := SEL(iOven = 2, Plant.fbSt010OvenA.OvenPickUpDepthZ, Plant.fbSt020OvenB.OvenPickUpDepthZ)
				+ fApprox;
END_GET
END_PROPERTY

{attribute 'monitoring' := 'call'}
PROPERTY PRIVATE PosWorkStorageX : LREAL
GET
PosWorkStorageX := SEL(stSt030IHandling.ActiveCommand.Position = 2,
						stSettings.stStationSettings[E_Station.eStation_ST040_Storage].stDynStationSettings[E_St040_Settings.eSt040_Settings_XPosStor1].fValue, 
						stSettings.stStationSettings[E_Station.eStation_ST040_Storage].stDynStationSettings[E_St040_Settings.eSt040_Settings_XPosStor2].fValue);
END_GET
END_PROPERTY

{attribute 'monitoring' := 'call'}
PROPERTY PRIVATE PosWorkStorageY : LREAL
GET
PosWorkStorageY := SEL(stSt030IHandling.ActiveCommand.Position = 2,
						stSettings.stStationSettings[E_Station.eStation_ST040_Storage].stDynStationSettings[E_St040_Settings.eSt040_Settings_YPosStor1].fValue,
						stSettings.stStationSettings[E_Station.eStation_ST040_Storage].stDynStationSettings[E_St040_Settings.eSt040_Settings_YPosStor2].fValue);
END_GET
END_PROPERTY

{attribute 'monitoring' := 'call'}
PROPERTY PRIVATE PosWorkStorageY_OffsDn : LREAL
GET
PosWorkStorageY_OffsDn := PosWorkStorageY - 15;//P_Plant.StorageOffsetDnY;
END_GET
END_PROPERTY

{attribute 'monitoring' := 'call'}
PROPERTY PRIVATE PosWorkStorageY_OffsUp : LREAL
GET
PosWorkStorageY_OffsUp := PosWorkStorageY + 20;// P_Plant.StorageOffsetUpY;
END_GET
END_PROPERTY

{attribute 'monitoring' := 'call'}
PROPERTY PRIVATE PosWorkStorageZ : LREAL
GET
PosWorkStorageZ := SEL(stSt030IHandling.ActiveCommand.Position = 2,
						stSettings.stStationSettings[E_Station.eStation_ST040_Storage].stDynStationSettings[E_St040_Settings.eSt040_Settings_ZPosStor1].fValue,
						stSettings.stStationSettings[E_Station.eStation_ST040_Storage].stDynStationSettings[E_St040_Settings.eSt040_Settings_ZPosStor2].fValue);
END_GET
END_PROPERTY

/// Reset station logic
{attribute 'object_name' := 'Reset'}
METHOD Reset
VAR
END_VAR
// base logic run
SUPER^.Reset();

// reset objects

IF fbAxisX.bError OR NOT RunCycle THEN
	fbAxisX.Reset();
END_IF
IF fbAxisY.bError OR NOT RunCycle THEN
	fbAxisY.Reset();
END_IF
IF fbAxisZ.bError OR NOT RunCycle THEN
	fbAxisZ.Reset();
END_IF
END_METHOD

{attribute 'monitoring' := 'call'}
PROPERTY PRIVATE WorkSpeedX : LREAL
GET
WorkSpeedX := stLocalSettings.stDynStationSettings[E_St030_Settings.eSt030_Settings_XWorkSpeed].fValue;
END_GET
END_PROPERTY

{attribute 'monitoring' := 'call'}
PROPERTY PRIVATE WorkSpeedY : LREAL
GET
WorkSpeedY := stLocalSettings.stDynStationSettings[E_St030_Settings.eSt030_Settings_YWorkSpeed].fValue;
END_GET
END_PROPERTY

{attribute 'monitoring' := 'call'}
PROPERTY PRIVATE WorkSpeedZ : LREAL
GET
WorkSpeedZ := stLocalSettings.stDynStationSettings[E_St030_Settings.eSt030_Settings_ZWorkSpeed].fValue;
END_GET
END_PROPERTY

END_FUNCTION_BLOCK

// ---- POUs/System/Utilities/FB_RtrigFtrig.TcPOU
FUNCTION_BLOCK PUBLIC FB_RtrigFtrig
VAR_INPUT
	bIn : BOOL;
END_VAR
VAR_OUTPUT
	// rising trigger bIn
	bRq : BOOL;
	// falling trigger bIn
	bFq : BOOL;
END_VAR
VAR
	rtrig : R_TRIG;
	ftrig : F_TRIG;
END_VAR

rtrig(CLK := bIn, Q => bRq);
ftrig(CLK := bIn, Q => bFq);

END_FUNCTION_BLOCK

// ---- POUs/Plant/ST040_Storage/FB_St040_Storage.TcPOU
FUNCTION_BLOCK FB_St040_Storage EXTENDS FB_StationBase
VAR_INPUT
END_VAR
VAR	
	// IO ref
	stIO			: REFERENCE TO ST_St040_IO;
	
	// station components
	fbAxis1,
	fbAxis2			: FB_AxisDriver;
	
	// actor UIs, access to: iStatus, fPosition, iVisibleState, ..
	fbAxis1Ui,
	fbAxis2Ui		: FB_Axis_Ui;
	
	// instance var's
	bStationDeaktiv	: BOOL;
END_VAR

/// 
/// Station 040 function block 
///

{attribute 'monitoring' := 'call'}
PROPERTY PRIVATE JogSpeed : LREAL
GET
JogSpeed := stLocalSettings.stDynStationSettings[E_St040_Settings.eSt040_Settings_JogSpeed].fValue;
END_GET
END_PROPERTY

METHOD PROTECTED M_CallObjects : BOOL
VAR_INPUT
END_VAR
// axis 1 + UI
fbAxis1(
	bEnable := SafetyOk AND NOT fbAxis1Ui.stAxisManager.bDisable,
	bEnablePos := TRUE,
	bEnableNeg := TRUE,
);
fbAxis1Ui(
	bInHome := bInHome,
	fbAxis := fbAxis1,
	fVelocity := JogSpeed,
	diSelectedObjectIndex := stHmiManualIn.diSelectedObjectIndex,
	stHMIControlIn := stHmiManualIn.stManualAxis,
	stHMIControlOut := stHmiManualOut.stManualAxis,
	bJogP := stHmi.stIn.stSt040.bJog01Up,
	bJogN := stHmi.stIn.stSt040.bJog01Down,
	bEnableManual := EnableManual);

// axis 2 + UI
fbAxis2(
	bEnable := SafetyOk AND NOT fbAxis2Ui.stAxisManager.bDisable,
	bEnablePos := TRUE,
	bEnableNeg := TRUE,
);
fbAxis2Ui(
	bInHome := bInHome,
	fbAxis := fbAxis2,
	fVelocity := JogSpeed,
	diSelectedObjectIndex := stHmiManualIn.diSelectedObjectIndex,
	stHMIControlIn := stHmiManualIn.stManualAxis,
	stHMIControlOut := stHmiManualOut.stManualAxis,
	bJogP := stHmi.stIn.stSt040.bJog02Up,
	bJogN := stHmi.stIn.stSt040.bJog02Down,
	bEnableManual := EnableManual);
	
// HMI : switch between jo modes
//IF stHmi.stIn.stSt040.bJog THEN
//	fbAxis1Ui.ManualMode :=  SEL(stHmi.stIn.stSt040.bSpeed, E_ManualMode.eManualMode_Jog01, E_ManualMode.eManualMode_Jog1);
//	fbAxis2Ui.ManualMode :=  SEL(stHmi.stIn.stSt040.bSpeed, E_ManualMode.eManualMode_Jog01, E_ManualMode.eManualMode_Jog1);
//ELSE
//	fbAxis1Ui.ManualMode :=  E_ManualMode.eManualMode_Tippen;//		SEL(stHmi.stIn.stSt030.bSpeed, E_ManualMode.eManualMode_TippSlow, E_ManualMode.eManualMode_TippFast);
//	fbAxis2Ui.ManualMode :=  E_ManualMode.eManualMode_Tippen;//		SEL(stHmi.stIn.stSt030.bSpeed, E_ManualMode.eManualMode_TippSlow, E_ManualMode.eManualMode_TippFast);
//END_IF		

// run pallet logic
//Plant.stSt040IStorage.Pallet1();
//Plant.stSt040IStorage.Pallet1.Update();
//Plant.stSt040IStorage.Pallet2();
//Plant.stSt040IStorage.Pallet2.Update();
END_METHOD

METHOD INTERNAL M_DynManual : BOOL
VAR_INPUT
END_VAR
IF NOT bInitManual THEN
	bInitManual := TRUE;
	MEMSET(ADR(stHmiManualOut.stObjects), 0, SIZEOF(stHmiManualOut.stObjects)); // reset
	
	M_InitDynManualUi(fbAxis1Ui);
	M_InitDynManualUi(fbAxis2Ui);
END_IF
END_METHOD

METHOD PROTECTED M_DynMonitoring : BOOL
VAR_INPUT
END_VAR
M_DynMonitoring := SUPER^.M_DynMonitoring();

// init
IF NOT bInitMonitoring THEN
	bInitMonitoring := TRUE;
	MEMSET(ADR(stLocalMonitoring), 0, SIZEOF(stLocalMonitoring)); // reset
	
	M_InitDynMonitoringItem(0, 								// monitoring index 
							"Achse 1 Position",				// name
							Name, 							// group (station name)
							E_DataType.eDataType_lreal, 	// data type							
							stTextListGlobal.stText_mm);	// unit	

	M_InitDynMonitoringItem(1, "Achse 1 Geschwindigkeit", Name, E_DataType.eDataType_lreal, stTextListGlobal.stText_mms);
	M_InitDynMonitoringItem(2, "Achse 1 Drehmoment", Name, E_DataType.eDataType_lreal, stTextListGlobal.stText_percent);
	
	M_InitDynMonitoringItem(4, "Achse 2 Position", Name, E_DataType.eDataType_lreal, stTextListGlobal.stText_mm);
	M_InitDynMonitoringItem(5, "Achse 2 Geschwindigkeit", Name, E_DataType.eDataType_lreal, stTextListGlobal.stText_mms);
	M_InitDynMonitoringItem(6, "Achse 2 Drehmoment", Name, E_DataType.eDataType_lreal, stTextListGlobal.stText_percent);
END_IF

// live value mapping 

// axis 1
stLocalMonitoring.astMonitoring[0].fValue := fbAxis1.Position;
stLocalMonitoring.astMonitoring[1].fValue := fbAxis1.Velocity;
stLocalMonitoring.astMonitoring[2].fValue := fbAxis1.Torque;

// axis 2
stLocalMonitoring.astMonitoring[4].fValue := fbAxis2.Position;
stLocalMonitoring.astMonitoring[5].fValue := fbAxis2.Velocity;
stLocalMonitoring.astMonitoring[6].fValue := fbAxis2.Torque;

// hmi value mapping
//HMI.stHmi.stOut.stSt040.Pallet1 := stSt040IStorage.Pallet1.stPallet;
//HMI.stHmi.stOut.stSt040.Pallet2 := stSt040IStorage.Pallet2.stPallet;
END_METHOD

METHOD INTERNAL M_DynSettings : BOOL
VAR_INPUT
END_VAR
// init station settings
IF NOT bInitSettings THEN
	bInitSettings := TRUE;
	stLocalSettingsBackup := stLocalSettings; // backup
	MEMSET(ADR(stLocalSettings), 0, SIZEOF(stLocalSettings)); // reset
	
	stSt040IStorage.Pallet1.Config := Services.stSettings.stCarrier;
	stSt040IStorage.Pallet1.InitialStatus := eTcaWorkpieceStatus.laserProcessDone;
	stSt040IStorage.Pallet1.RequestStatus := eTcaWorkpieceStatus.castingProcessDone;
	stSt040IStorage.Pallet1.ApplyConfig();
	     
	stSt040IStorage.Pallet2.Config := Services.stSettings.stCarrier;
	stSt040IStorage.Pallet2.InitialStatus := eTcaWorkpieceStatus.laserProcessDone;
	stSt040IStorage.Pallet2.RequestStatus := eTcaWorkpieceStatus.castingProcessDone;
	stSt040IStorage.Pallet2.ApplyConfig();
	
	
	M_InitDynSettingsItem(E_St040_Settings.eSt040_Settings_Station_Deaktiv,	// settings index
		TO_WSTRING(E_St040_Settings.eSt040_Settings_Station_Deaktiv),		// settings wsIndex
		Name,																// group
		stTextListGlobal.stText_DeactivateStation,							// name
		stTextListGlobal.stText_bool, E_DataType.eDataType_bool,			// unit & data type
		0, 1, 3);															// min, max & user level

	M_InitDynSettingsItem(E_St040_Settings.eSt040_Settings_Autohome,
		TO_WSTRING(E_St040_Settings.eSt040_Settings_Autohome),
		Name,
		stTextListGlobal.stText_AutoHome,
		stTextListGlobal.stText_bool, E_DataType.eDataType_bool,
		0, 1, 3);

	M_InitDynSettingsItem(E_St040_Settings.eSt040_Settings_JogSpeed,
		TO_WSTRING(E_St040_Settings.eSt040_Settings_JogSpeed),
		Name,
		F_CreateDynTextDefault("Tippgeschwindigkeit Servoachse"),
		stTextListGlobal.stText_mms, E_DataType.eDataType_lreal,
		0, 50, 3);
		
	M_InitDynSettingsItem(E_St040_Settings.eSt040_Settings_WorkSpeed,
		TO_WSTRING(E_St040_Settings.eSt040_Settings_WorkSpeed),
		Name,
		F_CreateDynTextDefault("Automatik-Geschwindigkeit Servoachse"),
		stTextListGlobal.stText_mms, E_DataType.eDataType_lreal,
		0, 500, 3);
		
	M_InitDynSettingsItem(E_St040_Settings.eSt040_Settings_PosHome,
		TO_WSTRING(E_St040_Settings.eSt040_Settings_PosHome),
		Name,
		F_CreateDynTextDefault("Homeposition Servoachse"),
		stTextListGlobal.stText_mm, E_DataType.eDataType_lreal,
		0, 500, 3);
		
	M_InitDynSettingsItem(E_St040_Settings.eSt040_Settings_PosWork,
		TO_WSTRING(E_St040_Settings.eSt040_Settings_PosWork),
		Name,
		F_CreateDynTextDefault("Arbeitsposition Servoachse"),
		stTextListGlobal.stText_mm, E_DataType.eDataType_lreal,
		0, 500, 3);

	M_InitDynSettingsItem(E_St040_Settings.eSt040_Settings_XPosStor1,	// Teach-Position, Storage 1 [mm]
		TO_WSTRING(E_St040_Settings.eSt040_Settings_XPosStor1),
		Name,
		F_CreateDynTextDefault("Teach-Position, Storage 1 X"),
		stTextListGlobal.stText_mm, E_DataType.eDataType_lreal,
		0, 5000, 3);
	M_InitDynSettingsItem(E_St040_Settings.eSt040_Settings_YPosStor1,
		TO_WSTRING(E_St040_Settings.eSt040_Settings_YPosStor1),
		Name,
		F_CreateDynTextDefault("Teach-Position, Storage 1 Y"),
		stTextListGlobal.stText_mm, E_DataType.eDataType_lreal,
		0, 5000, 3);
	M_InitDynSettingsItem(E_St040_Settings.eSt040_Settings_ZPosStor1,
		TO_WSTRING(E_St040_Settings.eSt040_Settings_ZPosStor1),
		Name,
		F_CreateDynTextDefault("Teach-Position, Storage 1 Z"),
		stTextListGlobal.stText_mm, E_DataType.eDataType_lreal,
		0, 5000, 3);
		
	M_InitDynSettingsItem(E_St040_Settings.eSt040_Settings_XPosStor2,	// Teach-Position, Storage 2 [mm]
		TO_WSTRING(E_St040_Settings.eSt040_Settings_XPosStor2),
		Name,
		F_CreateDynTextDefault("Teach-Position, Storage 2 X"),
		stTextListGlobal.stText_mm, E_DataType.eDataType_lreal,
		0, 5000, 3);
	M_InitDynSettingsItem(E_St040_Settings.eSt040_Settings_YPosStor2,
		TO_WSTRING(E_St040_Settings.eSt040_Settings_YPosStor2),
		Name,
		F_CreateDynTextDefault("Teach-Position, Storage 2 Y"),
		stTextListGlobal.stText_mm, E_DataType.eDataType_lreal,
		0, 5000, 3);
	M_InitDynSettingsItem(E_St040_Settings.eSt040_Settings_ZPosStor2,
		TO_WSTRING(E_St040_Settings.eSt040_Settings_ZPosStor2),
		Name,
		F_CreateDynTextDefault("Teach-Position, Storage 2 Z"),
		stTextListGlobal.stText_mm, E_DataType.eDataType_lreal,
		0, 5000, 3);

		
	// restore values
	F_RestoreSettingValues(stLocalSettings.stDynStationSettings, stLocalSettingsBackup.stDynStationSettings);
END_IF

// map current settings values
bAutoHome := stLocalSettings.stDynStationSettings[E_St040_Settings.eSt040_Settings_Autohome].bValue;
bStationDeaktiv := stLocalSettings.stDynStationSettings[E_St040_Settings.eSt040_Settings_Station_Deaktiv].bValue;
END_METHOD

METHOD PROTECTED M_Homing
VAR
END_VAR
// Homing sequence
CASE sqHome.Step OF
	
	0:	
		sqHome.Info.Set("Warte auf GRST Start");
		IF RunStep AND NOT sqHome.InHome AND bRunHoming THEN
			bBusy := TRUE;
			sqAuto.Step := 0;
			sqHome.StartSequence()
				  .Step := 10;
		END_IF

	10:
		sqHome.Info.Set("Grundstellungsfahrt aktiv");
		IF P_Safety.bMachineRequestStop THEN
			sqHome.Info.Set("Anforderung Stop aktiv");
		ELSIF NOT P_Safety.EmergencyStopOk THEN
			sqHome.Info.Set("Sicherheit nicht ok");
			
		ELSIF NOT fbAxis1.Operational THEN
			sqHome.Info.Set("Antrieb 1 nicht bereit");
		ELSIF fbAxis1.Moving THEN
			fbAxis1.Halt();
			sqHome.Info.Set("Antrieb 1 nicht gestoppt");
			
		ELSIF NOT fbAxis2.Operational THEN
			sqHome.Info.Set("Antrieb 2 nicht bereit");
		ELSIF fbAxis2.Moving THEN
			fbAxis2.Halt();
			sqHome.Info.Set("Antrieb 2 nicht gestoppt");

		ELSIF bRunHoming THEN
			sqHome.SetStep(20);
		END_IF	
		
	20:
		sqHome.Info.Set("Grundstellungsfahrt aktiv Achse 1/2 auf Homepos.");
		fbAxis1.MoveAbsExVel(PosHome, WorkSpeed);
		fbAxis2.MoveAbsExVel(PosHome, WorkSpeed);
		sqHome.Step := 25;
		
	25:
		sqHome.Info.Set("Warte auf Achse 1 in Homeposition");
		IF NOT fbAxis1.TargetWindowReached(chAxisPosTol + 4) THEN RETURN; END_IF //ToDo: set pos tol
		sqHome.Info.Set("Warte auf Achse 2 in Homeposition");
		IF NOT fbAxis2.TargetWindowReached(chAxisPosTol + 4) THEN RETURN; END_IF //ToDo: set pos tol
		sqHome.Step := 100;
		
	100:
		sqHome.Info.Set("Grundstellungsfahrt aktiv");
		sqHome.Step := 1000;

	//	homing done			
	1000:
		sqHome.Info.Set("Grundstellung erreicht");
		IF sqHome.StepTime > T#1S THEN
			bBusy:=FALSE;
			sqHome.InHome := TRUE;
			bStopped := TRUE;
			bRunHoming := FALSE;
			sqAuto.Step := 0;
			sqHome.StopSequence()
				  .Step := 0;
		END_IF
END_CASE
END_METHOD

METHOD PUBLIC M_Init : IStation
VAR_INPUT
END_VAR
VAR
	Ist : IStation;
END_VAR
// set up station
StationNb := 40;
Station := E_Station.eStation_ST040_Storage; // ID & name 1st!
Name := F_CreateDynTextEx(1, "ST040_Storage", "ST040 Storage");

Ist := SUPER^.M_Init()
			 .InitEvents(TC_Events.ST040EventClass.InfoEvent,
	  		       		 TC_Events.ST040EventClass.WarningEvent,
	  				  	 TC_Events.ST040EventClass.ErrorEvent);

// set up default IO references
M_SetReferences(IO.st040_Storage_IO);

// init components

// Axis 1
fbAxis1Ui.stBmk := F_CreateDynTextDefault("BMK=A03.ST40.M01-");
fbAxis1Ui.stUnit := F_CreateDynTextDefault("mm");
fbAxis1Ui.stAxisManager.bEnablePosSet := TRUE;
fbAxis1.AxisId := TO_INT(E_Axis.eAxis_Storage1);
fbAxis1.Active := TRUE;
fbAxis1.Name := F_CreateDynTextEx(1, "Servo1", "Servoachse 1");
fbAxis1.AxisType := E_AxisType.AX5xxx;
//fbAxis1.DefaultParameter := F_GetDefaultMotionParameter(eMainState_setup);
fbAxis1.SetAxisReference(NcIO.stAxis_ST040_Axis1, NcIO.stAxis_ST040_Axis1_IO.stIn, NCIO.stAxis_ST040_Axis1_IO.stOut);

// Axis 2
fbAxis2Ui.stBmk := F_CreateDynTextDefault("BMK=A03.ST40.M02-");
fbAxis2Ui.stUnit := F_CreateDynTextDefault("mm");
fbAxis2Ui.stAxisManager.bEnablePosSet := TRUE;
fbAxis2.AxisId := TO_INT(E_Axis.eAxis_Storage2);
fbAxis2.Active := TRUE;
fbAxis2.Name := F_CreateDynTextEx(1, "Servo2", "Servoachse 2");
fbAxis2.AxisType := E_AxisType.AX5xxx;
//fbAxis2.DefaultParameter := F_GetDefaultMotionParameter(eMainState_setup);
fbAxis2.SetAxisReference(NcIO.stAxis_ST040_Axis2, NcIO.stAxis_ST040_Axis2_IO.stIn, NCIO.stAxis_ST040_Axis2_IO.stOut);

// register station in it's module
eParent := fbModul001.M_RegisterStation(Ist);

bInitSettings	:= FALSE;
bInitMonitoring := FALSE;
bInitManual  	:= FALSE;

//aSClearText[EN] := 'Station init done.';
M_Init := Ist;
END_METHOD

METHOD PROTECTED M_Manual
VAR
	fbPL : REFERENCE TO TcaCarrier;
END_VAR

// station must be stopped!			manual mode
IF RunCycle OR NOT bStopped THEN //(OpMode <> E_OpMode.eOpMode_manual) THEN
	RETURN;
END_IF

//IF stHmiInOut.stSt040.Command = E_HMI_PL_CMD.eHmiPlCmd_none AND_THEN 
//   stHmiInOut.stSt040.WpCmd.Command <> E_HMI_WP_CMD.eHmiWpCmd_none THEN
//	stHmiInOut.stSt040.Command := E_HMI_PL_CMD.eHmiPlCmd_performWtCmd;
//END_IF
//
//IF stHmiInOut.stSt040.Command = E_HMI_PL_CMD.eHmiPlCmd_none THEN
//	RETURN;
//END_IF

//IF stHmiInOut.stSt040.Idx = 1 THEN
//	fbPL REF= stSt040IStorage.Pallet1;
//ELSIF stHmiInOut.stSt040.Idx = 2 THEN
//	fbPL REF= stSt040IStorage.Pallet2;
//ELSE
//	StationError.ArgSbAppendRaise('Index not set on HMI Pallet Command');
//	//stHmiInOut.stSt040.Command := E_HMI_PL_CMD.eHmiPlCmd_none;
//	RETURN;
//END_IF

//fbPL.PerformHmiCmd(stHmiInOut.stSt040);
END_METHOD

METHOD PROTECTED M_OpModeChanged : BOOL
VAR_INPUT
END_VAR
(*bBusy := FALSE;

IF (eOpMode <> eOpMode_step AND eOpMode <> eOpMode_auto) THEN
	sqAuto.Set(0);
END_IF

fbAxis1.Stop();
fbAxis2.Stop();*)
END_METHOD

METHOD PUBLIC M_Run : BOOL
VAR_INPUT
END_VAR
// check refs valid
IF NOT __ISVALIDREF(stIO) THEN
	RETURN;
END_IF

M_RUN := SUPER^.M_Run();

M_DynSettings();
M_DynManual();
M_DynMonitoring();
END_METHOD

METHOD PROTECTED M_Sequence
VAR
END_VAR
// signal mapping (e.g.: enable)
// stSt040Interface.bEnable := (sqAuto.Step = 100 AND fbAxis1.Operational AND fbAxis1.Operational) OR
// 								bStationDeaktiv;

// automatic sequence
CASE sqAuto.Step OF
	
	0:	sqAuto.Info.Set("Warte auf Auto Start");
		IF RunCycle AND RunStep THEN
			//sqAuto.Info.Set("Warte auf GRST");
			//IF sqHome.InHome AND bInHome THEN
				sqHome.InHome := FALSE;
				sqAuto.Step := 5;
			//ELSE
			//	StationError.ArgSbAppendWsRaise(stTextlistGlobal.stText_station_not_in_hp);
			//END_IF
		END_IF
		
	5:	IF bStationDeaktiv THEN
			sqAuto.Info.Set("Station deaktiv");
		ELSE
			sqAuto.Step := 10;
		END_IF
		
	10:	sqAuto.Info.Set("Prüfe Startbedingungen");
		IF NOT fbAxis1.Operational THEN
			StationError.ArgSbAppendRaise('Bereitsignal Achse 1 fehlt');
		ELSIF NOT fbAxis2.Operational THEN
			StationError.ArgSbAppendRaise('Bereitsignal Achse 2 fehlt');
		ELSE
			CycleStart();
			sqAuto.SetStep(20);
		END_IF
		
	20:
		sqAuto.Info.Set("Automatik, Achse 1/2 auf Homepos.");
		fbAxis1.MoveAbsExVel(PosHome, WorkSpeed);
		fbAxis2.MoveAbsExVel(PosHome, WorkSpeed);
		sqAuto.Step := 25;
		
	25:
		sqAuto.Info.Set("Warte auf Achse 1 in Homeposition");
		IF NOT fbAxis1.TargetWindowReached(chAxisPosTol + 4) THEN RETURN; END_IF //ToDo: set pos tol
		sqAuto.Info.Set("Warte auf Achse 2 in Homeposition");
		IF NOT fbAxis2.TargetWindowReached(chAxisPosTol + 4) THEN RETURN; END_IF //ToDo: set pos tol
		sqAuto.Step := 100;

	// work
	100: sqAuto.Info.Set("Automatik, warte auf Anforderung vom HG");
		IF stSt030IHandling.bReqestStorage_ChkIndex THEN
			sqAuto.Info.Append(", Index-Check");
			stSt040IStorage.iConfirmPosition := stSt030IHandling.ActiveCommand.Position;
			//stSt040IStorage.iConfirmOpnIdxY := stSt030IHandling.ActiveCommand.IndexY;
			stSt040IStorage.bResponseEmptyAtIndex := (stSt030IHandling.ActiveCommand.Position = 1 AND NOT stSt040IStorage.Pallet1.CarrierPresent) OR
													 (stSt030IHandling.ActiveCommand.Position = 2 AND NOT stSt040IStorage.Pallet2.CarrierPresent);
			stSt040IStorage.bResponseChkIndex := TRUE;
			IF stSt030IHandling.bReqestStorage AND stSt040IStorage.iConfirmPosition = 1 THEN sqAuto.SetStep(110); END_IF
			IF stSt030IHandling.bReqestStorage AND stSt040IStorage.iConfirmPosition = 2 THEN sqAuto.SetStep(120); END_IF
		END_IF
	
		IF RunCycle THEN RETURN; END_IF
		sqAuto.Info.Set("Stop - warte auf Ablauf gestoppt");
		sqAuto.Step := 900;
		
	110:
		sqAuto.Info.Set("Automatik, Achse 1 öffnen");
		fbAxis1.MoveAbsExVel(PosHome, WorkSpeed);
		sqAuto.Step := 115;
		
	115:
		sqAuto.Info.Set("Warte auf Achse 1 Offenpos.");
		IF NOT fbAxis1.TargetWindowReached(chAxisPosTol + 4) THEN RETURN; END_IF //ToDo: set pos tol
		sqAuto.Step := 150;
		
	120:
		sqAuto.Info.Set("Automatik, Achse 2 öffnen");
		fbAxis2.MoveAbsExVel(PosHome, WorkSpeed);
		sqAuto.Step := 125;
		
	125:
		sqAuto.Info.Set("Warte auf Achse 2 in Offenpos.");
		IF NOT fbAxis2.TargetWindowReached(chAxisPosTol + 4) THEN RETURN; END_IF //ToDo: set pos tol
		sqAuto.Step := 150;
		
	150: sqAuto.Info.Set("Storage offen, warte auf Anforderung vom HG");
		stSt040IStorage.bResponseOpn := TRUE;
		IF NOT stSt030IHandling.bReqestStorage THEN
			stSt040IStorage.bResponseOpn := FALSE;
			sqAuto.SetStep(900);
		END_IF
		
	// rdy	
	900: sqAuto.Info.Set("Zyklus beendet");
		CycleEnd();
		sqAuto.Step := 0;

	// error
	1000: sqAuto.Info.Set("Error");
		bStopped := TRUE;
		sqHome.InHome := FALSE;
		bRunHoming := FALSE;

END_CASE
END_METHOD

METHOD INTERNAL M_SetReferences : BOOL
VAR_IN_OUT
	stIoRef : ST_St040_IO;
END_VAR
stIO REF= stIoRef;
M_SetReferences := TRUE;
END_METHOD

METHOD PROTECTED M_Supervision : BOOL
VAR_INPUT
END_VAR
// chk stopped
IF NOT bRunCycle OR P_Safety.bMachineRequestStop THEN
	IF sqAuto.StepTime > T#20S THEN
		bStopped := TRUE;
	END_IF
END_IF

// chk requested index
IF stSt030IHandling.bReqestStorage_ChkIndex THEN
	;// --> confirm chk implemented in M_Sequence, step 100
	//stSt040IStorage.iConfirmOpnIdx := stSt030IHandling.ActiveCommand.IndexX;
	////stSt040IStorage.iConfirmOpnIdxY := stSt030IHandling.ActiveCommand.IndexY;
	//stSt040IStorage.bResponseEmptyAtIndex := (stSt030IHandling.ActiveCommand.IndexX = 1 AND NOT stSt040IStorage.Pallet1.PalletExists) OR
	//										 (stSt030IHandling.ActiveCommand.IndexX = 2 AND NOT stSt040IStorage.Pallet2.PalletExists);
	//stSt040IStorage.bResponseChkIndex := TRUE;
ELSE
	stSt040IStorage.iConfirmPosition := -1;
	//stSt040IStorage.iConfirmOpnIdxY := -1;
	stSt040IStorage.bResponseEmptyAtIndex := FALSE;
	stSt040IStorage.bResponseChkIndex := FALSE;
END_IF

// axis x
IF fbAxis1.bError THEN
	ReactToComponentError(fbAxis1Ui, E_EventReaction.Stop);

// y
ELSIF fbAxis2.bError THEN
	ReactToComponentError(fbAxis2Ui, E_EventReaction.Stop);
	
END_IF
END_METHOD

{attribute 'monitoring' := 'call'}
PROPERTY PRIVATE PosHome : LREAL
GET
PosHome := stLocalSettings.stDynStationSettings[E_St040_Settings.eSt040_Settings_PosHome].fValue;
END_GET
END_PROPERTY

{attribute 'monitoring' := 'call'}
PROPERTY PRIVATE PosWork : LREAL
GET
PosWork := stLocalSettings.stDynStationSettings[E_St040_Settings.eSt040_Settings_PosWork].fValue;
END_GET
END_PROPERTY

/// Reset station logic
{attribute 'object_name' := 'Reset'}
METHOD Reset
VAR
END_VAR
// base logic run
SUPER^.Reset();

// reset objects

IF fbAxis1.bError OR NOT RunCycle THEN
	fbAxis1.Reset();
END_IF
IF fbAxis2.bError OR NOT RunCycle THEN
	fbAxis2.Reset();
END_IF
END_METHOD

{attribute 'monitoring' := 'call'}
PROPERTY PRIVATE WorkSpeed : LREAL
GET
WorkSpeed := stLocalSettings.stDynStationSettings[E_St040_Settings.eSt040_Settings_WorkSpeed].fValue;
END_GET
END_PROPERTY

END_FUNCTION_BLOCK

// ---- POUs/Plant/ST050_Mould/FB_St050_Mould.TcPOU
FUNCTION_BLOCK FB_St050_Mould EXTENDS FB_StationBase
VAR_INPUT
END_VAR
VAR	
	// IO ref
	stIO			: REFERENCE TO ST_St050_IO;
	
	stFromEngel 	: TcaEngelCastingCarrierInput;
	stToEngel 		: TcaEngelCastingCarrierOutput;
	
	// station components
	fbCamAs 		: FB_Device;
	fbCamBs 		: FB_Device;
	fbLedAs 		: FB_Device;
	fbLedBs 		: FB_Device;
	
	// actor UIs, access to: iStatus, fPosition, iVisibleState, ..
	fbCamAsUi 		: FB_Device_Ui;
	fbCamBsUi 		: FB_Device_Ui;
	fbLedAsUi 		: FB_Device_Ui;
	fbLedBsUi 		: FB_Device_Ui;
	
	// instance var's
	bStationDeaktiv	: BOOL;
END_VAR

/// 
/// Station 060 function block 
///

METHOD PROTECTED M_CallObjects : BOOL
VAR_INPUT
END_VAR
// Cam's + UI
fbCamAs.Enable := P_Safety.EmergencyStopOk;
//fbCamAs.Value := stLocalSettings.stDynStationSettings[E_St060_Settings.eSt060_Settings_CamPrgAs].nValue;
fbCamAs();
fbCamAsUi(diSelectedObjectIndex := stHmiManualIn.diSelectedObjectIndex,
	stHMIControlIn := stHmiManualIn.stManualDevice,
	stHMIControlOut := stHmiManualOut.stManualDevice,
	fbDevice := fbCamAs,
	bEnableManual := EnableManual);
	
fbCamBs.Enable := P_Safety.EmergencyStopOk;
//fbCamBs.Value := stLocalSettings.stDynStationSettings[E_St060_Settings.eSt060_Settings_CamPrgBs].nValue;
fbCamBs();
fbCamBsUi(diSelectedObjectIndex := stHmiManualIn.diSelectedObjectIndex,
	stHMIControlIn := stHmiManualIn.stManualDevice,
	stHMIControlOut := stHmiManualOut.stManualDevice,
	fbDevice := fbCamBs,
	bEnableManual := EnableManual);
	
// LED's + UI
fbLedAs.Enable := P_Safety.EmergencyStopOk;
fbLedAs();
fbLedAsUi(diSelectedObjectIndex := stHmiManualIn.diSelectedObjectIndex,
	stHMIControlIn := stHmiManualIn.stManualDevice,
	stHMIControlOut := stHmiManualOut.stManualDevice,
	fbDevice := fbLedAs,
	bEnableManual := EnableManual);
	
fbLedBs.Enable := P_Safety.EmergencyStopOk;
fbLedBs();
fbLedBsUi(diSelectedObjectIndex := stHmiManualIn.diSelectedObjectIndex,
	stHMIControlIn := stHmiManualIn.stManualDevice,
	stHMIControlOut := stHmiManualOut.stManualDevice,
	fbDevice := fbLedBs,
	bEnableManual := EnableManual);
END_METHOD

METHOD INTERNAL M_DynManual : BOOL
VAR_INPUT
END_VAR
IF NOT bInitManual THEN
	bInitManual := TRUE;
	MEMSET(ADR(stHmiManualOut.stObjects), 0, SIZEOF(stHmiManualOut.stObjects)); // reset
	
	//M_InitDynManualUi(fbObjectUi);
END_IF

// additional states
END_METHOD

METHOD PROTECTED M_DynMonitoring : BOOL
VAR_INPUT
END_VAR
M_DynMonitoring := SUPER^.M_DynMonitoring();

// init
IF NOT bInitMonitoring THEN
	bInitMonitoring := TRUE;
	MEMSET(ADR(stLocalMonitoring), 0, SIZEOF(stLocalMonitoring)); // reset
	
	M_InitDynMonitoringItem(0, 								// monitoring index 
							"Engel SGM CycleMode", 			// name
							Name, 							// group (station name)
							E_DataType.eDataType_bool, 		// data type							
							stTextListGlobal.stText_bool);	// unit	
    
	M_InitDynMonitoringItem(1, "Engel SGM SequenceMode", Name, E_DataType.eDataType_bool, stTextListGlobal.stText_bool);
	M_InitDynMonitoringItem(2, "Engel SGM ProductionEnd", Name, E_DataType.eDataType_bool, stTextListGlobal.stText_bool);
	M_InitDynMonitoringItem(3, "Engel SGM Error", Name, E_DataType.eDataType_bool, stTextListGlobal.stText_bool);
	M_InitDynMonitoringItem(4, "Engel SGM ErrorID", Name, E_DataType.eDataType_int, stTextListGlobal.stText_notext);	
	M_InitDynMonitoringItem(5, "Engel SGM Moving", Name, E_DataType.eDataType_bool, stTextListGlobal.stText_bool);
	M_InitDynMonitoringItem(6, "Engel SGM ParkPosition", Name, E_DataType.eDataType_bool, stTextListGlobal.stText_bool);
	M_InitDynMonitoringItem(7, "Engel SGM SafetyAreaSafe", Name, E_DataType.eDataType_bool, stTextListGlobal.stText_bool);
	M_InitDynMonitoringItem(8, "Engel SGM OutsideStorage_1", Name, E_DataType.eDataType_bool, stTextListGlobal.stText_bool);
	M_InitDynMonitoringItem(9, "Engel SGM OutsideStorage_2", Name, E_DataType.eDataType_bool, stTextListGlobal.stText_bool);
END_IF

// live value mapping 
stLocalMonitoring.astMonitoring[0].bValue := stFromEngel.AutoMode;
stLocalMonitoring.astMonitoring[1].bValue := stFromEngel.SemiAutoMode;
stLocalMonitoring.astMonitoring[2].bValue := stFromEngel.ManualMode;
stLocalMonitoring.astMonitoring[3].bValue := stFromEngel.Error;
stLocalMonitoring.astMonitoring[4].nValue := stFromEngel.ErrorID;
stLocalMonitoring.astMonitoring[5].bValue := stFromEngel.Moving;
stLocalMonitoring.astMonitoring[6].bValue := stFromEngel.ParkPosition;
stLocalMonitoring.astMonitoring[7].bValue := stFromEngel.SafetyAreaSafe;
stLocalMonitoring.astMonitoring[8].bValue := stFromEngel.OutsideStorage_1;
stLocalMonitoring.astMonitoring[9].bValue := stFromEngel.OutsideStorage_2;
END_METHOD

METHOD INTERNAL M_DynSettings : BOOL
VAR_INPUT
END_VAR
// init station settings
IF NOT bInitSettings THEN
	bInitSettings := TRUE;
	stLocalSettingsBackup := stLocalSettings; // backup
	MEMSET(ADR(stLocalSettings), 0, SIZEOF(stLocalSettings)); // reset
	
	M_InitDynSettingsItem(E_St050_Settings.eSt050_Settings_Station_Deaktiv,	// settings index
		TO_WSTRING(E_St050_Settings.eSt050_Settings_Station_Deaktiv),		// settings wsIndex
		Name,																// group
		stTextListGlobal.stText_DeactivateStation,							// name
		stTextListGlobal.stText_bool, E_DataType.eDataType_bool,			// unit & data type
		0, 1, 3);															// min, max & user level

	M_InitDynSettingsItem(E_St050_Settings.eSt050_Settings_Autohome,
		TO_WSTRING(E_St050_Settings.eSt050_Settings_Autohome),
		Name,
		stTextListGlobal.stText_AutoHome,
		stTextListGlobal.stText_bool, E_DataType.eDataType_bool,
		0, 1, 3);
		
	(*M_InitDynSettingsItem(E_St060_Settings.eSt060_Settings_CamPrgAs,
		TO_WSTRING(E_St060_Settings.eSt060_Settings_CamPrgAs),
		Name,
		F_CreateDynTextDefault("Kammeraprogamm"),
		stTextListGlobal.stText_KameraProgramm, E_DataType.eDataType_int,
		1, 9999, 3);
	
	M_InitDynSettingsItem(E_St060_Settings.eSt060_Settings_CamPrgBs,
		TO_WSTRING(E_St060_Settings.eSt060_Settings_CamPrgBs),
		Name,
		F_CreateDynTextDefault("Kammeraprogamm"),
		stTextListGlobal.stText_KameraProgramm, E_DataType.eDataType_int,
		1, 9999, 3);
		
	M_InitDynSettingsItem(E_St060_Settings.eSt060_Settings_LedAs,
		TO_WSTRING(E_St060_Settings.eSt060_Settings_LedAs),
		Name,
		F_CreateDynTextDefault("LED AS"),
		stTextListGlobal.stText_bool, E_DataType.eDataType_bool,
		0, 1, 3);
		
	M_InitDynSettingsItem(E_St060_Settings.eSt060_Settings_LedBs,
		TO_WSTRING(E_St060_Settings.eSt060_Settings_LedBs),
		Name,
		F_CreateDynTextDefault("LED BS"),
		stTextListGlobal.stText_bool, E_DataType.eDataType_bool,
		0, 1, 3); *)
		
	// restore values
	F_RestoreSettingValues(stLocalSettings.stDynStationSettings, stLocalSettingsBackup.stDynStationSettings);
END_IF

// map current settings values
bAutoHome := stLocalSettings.stDynStationSettings[E_St050_Settings.eSt050_Settings_Autohome].bValue;
bStationDeaktiv := stLocalSettings.stDynStationSettings[E_St050_Settings.eSt050_Settings_Station_Deaktiv].bValue;
END_METHOD

METHOD PROTECTED M_Homing
VAR
END_VAR
// Homing sequence
CASE sqHome.Step OF
	
	0:	
		sqHome.Info.Set("Warte auf GRST Start");
		IF RunStep AND NOT sqHome.InHome AND bRunHoming THEN
			bBusy := TRUE;
			sqAuto.Step := 0;
			sqHome.StartSequence()
				  .Step := 10;
		END_IF

	10:
		sqHome.Info.Set("Grundstellungsfahrt aktiv");
		IF P_Safety.bMachineRequestStop THEN
			sqHome.Info.Set("Anforderung Stop aktiv");
		ELSIF NOT P_Safety.EmergencyStopOk THEN
			sqHome.Info.Set("Sicherheit nicht ok");
		//ELSIF NOT fbCamAs.bRdy THEN
		//	sqHome.Info.Set("Kamera AS nicht bereit");
		//ELSIF fbCamAs.bErr THEN
		//	sqHome.Info.Set("Kamera AS meldet Fehler");
		// ...

		ELSIF bRunHoming THEN
			sqHome.Step := 100;
		END_IF	
		
	100:
		sqHome.Info.Set("Grundstellungsfahrt aktiv");
		sqHome.Step := 1000;

	//	homing done			
	1000:
		sqHome.Info.Set("Grundstellung erreicht");
		IF sqHome.StepTime > T#1S THEN
			bBusy:=FALSE;
			sqHome.InHome := TRUE;
			bStopped := TRUE;
			bRunHoming := FALSE;
			sqAuto.Step := 0;
			sqHome.StopSequence()
				  .Step := 0;
		END_IF
END_CASE
END_METHOD

METHOD PUBLIC M_Init : IStation
VAR_INPUT
END_VAR
VAR
	Ist : IStation;
END_VAR
// set up station
StationNb := 50;
Station := E_Station.eStation_ST050_Mould; // ID & name 1st!
Name := F_CreateDynTextEx(1, "eStation_ST050_Mould", "ST050 Mould");

Ist := SUPER^.M_Init()
			 .InitEvents(TC_Events.ST050EventClass.InfoEvent,
	  		       		 TC_Events.ST050EventClass.WarningEvent,
	  				  	 TC_Events.ST050EventClass.ErrorEvent);

// set up default IO references
M_SetReferences(IO.St050_Mould_IO);

// init components

// Kameras & LEDs
fbCamAsUi.stBmk := F_CreateDynTextDefault("BMK=+xyz-");
fbCamAs.Active := TRUE;
fbCamAs.Name := F_CreateDynTextEx(1, "MouldKameraAs", "Engel SGM Kamera AS");

fbCamBsUi.stBmk := F_CreateDynTextDefault("BMK=ST52.B01.1BX1-");
fbCamBs.Active := TRUE;
fbCamBs.Name := F_CreateDynTextEx(1, "MouldKameraBs", "Engel SGM Kamera BS");

fbLedAsUi.stBmk := F_CreateDynTextDefault("BMK=+xyz-");
fbLedAs.Active := TRUE;
fbLedAs.Name := F_CreateDynTextEx(1, "MouldLedAs", "Engel SGM LED AS");

fbLedBsUi.stBmk := F_CreateDynTextDefault("BMK=+xyz-");
fbLedBs.Active := TRUE;
fbLedBs.Name := F_CreateDynTextEx(1, "MouldLedBs", "Engel SGM LED BS");


// register station in it's module
eParent := fbModul001.M_RegisterStation(Ist);

bInitSettings	:= FALSE;
bInitMonitoring := FALSE;
bInitManual  	:= FALSE;

//aSClearText[EN] := 'Station init done.';
M_Init := Ist;
END_METHOD

METHOD PROTECTED M_Manual
VAR
END_VAR

// manual mode
IF (OpMode <> E_OpMode.eOpMode_manual) THEN
	RETURN;
END_IF
END_METHOD

METHOD PRIVATE M_MappingIn : BOOL
VAR_INPUT
END_VAR
MEMCPY(ADR(stFromEngel.LifeCounter), ADR(stIo.stIn.aFromEngelRaw[0]), SIZEOF(UINT));
MEMCPY(ADR(stFromEngel.ErrorID), ADR(stIo.stIn.aFromEngelRaw[2]), SIZEOF(UINT));
RETURN;
stFromEngel.AutoMode := stIo.stIn.aFromEngelRaw[4].0;
stFromEngel.SemiAutoMode := stIo.stIn.aFromEngelRaw[4].1;
stFromEngel.ManualMode := stIo.stIn.aFromEngelRaw[4].2;
stFromEngel.Error := stIo.stIn.aFromEngelRaw[4].3;
stFromEngel.Moving := stIo.stIn.aFromEngelRaw[4].4;
stFromEngel.ParkPosition := stIo.stIn.aFromEngelRaw[4].5;
stFromEngel.OutsideStorage_1 := stIo.stIn.aFromEngelRaw[4].6;
stFromEngel.OutsideStorage_2 := stIo.stIn.aFromEngelRaw[4].7;

stFromEngel.SafetyAreaSafe := stIo.stIn.aFromEngelRaw[5].0;

stFromEngel.JobForStorage_1.RequestNoCarrier := stIo.stIn.aFromEngelRaw[5].1;
stFromEngel.JobForStorage_1.RequestCarrier := stIo.stIn.aFromEngelRaw[5].2;
stFromEngel.JobForStorage_1.Empty := stIo.stIn.aFromEngelRaw[5].3;
stFromEngel.JobForStorage_1.Unfinished := stIo.stIn.aFromEngelRaw[5].4;

stFromEngel.JobForStorage_2.RequestNoCarrier := stIo.stIn.aFromEngelRaw[5].5;
stFromEngel.JobForStorage_2.RequestCarrier := stIo.stIn.aFromEngelRaw[5].6;
stFromEngel.JobForStorage_2.Empty := stIo.stIn.aFromEngelRaw[5].7;

stFromEngel.JobForStorage_2.Unfinished := stIo.stIn.aFromEngelRaw[6].0;

//stFromEngel.Res. := stIo.stIn.aFromEngelRaw[6].1;
//...
//stFromEngel.Res. := stIo.stIn.aFromEngelRaw[6].7;

MEMCPY(ADR(stFromEngel.JobForStorage_1.CarrierId), ADR(stIo.stIn.aFromEngelRaw[7]), SIZEOF(UINT));
MEMCPY(ADR(stFromEngel.JobForStorage_2.CarrierId), ADR(stIo.stIn.aFromEngelRaw[9]), SIZEOF(UINT));

MEMCPY(ADR(stFromEngel.Storage_1.CarrierId), ADR(stIo.stIn.aFromEngelRaw[11]), SIZEOF(UINT));
MEMCPY(ADR(stFromEngel.Storage_1.CountMax), ADR(stIo.stIn.aFromEngelRaw[13]), SIZEOF(UINT));
MEMCPY(ADR(stFromEngel.Storage_1.CountUnfinished), ADR(stIo.stIn.aFromEngelRaw[15]), SIZEOF(UINT));
MEMCPY(ADR(stFromEngel.Storage_1.CountFinished), ADR(stIo.stIn.aFromEngelRaw[17]), SIZEOF(UINT));
MEMCPY(ADR(stFromEngel.Storage_1.CountEmpty), ADR(stIo.stIn.aFromEngelRaw[19]), SIZEOF(UINT));

MEMCPY(ADR(stFromEngel.Storage_2.CarrierId), ADR(stIo.stIn.aFromEngelRaw[21]), SIZEOF(UINT));
MEMCPY(ADR(stFromEngel.Storage_2.CountMax), ADR(stIo.stIn.aFromEngelRaw[23]), SIZEOF(UINT));
MEMCPY(ADR(stFromEngel.Storage_2.CountUnfinished), ADR(stIo.stIn.aFromEngelRaw[25]), SIZEOF(UINT));
MEMCPY(ADR(stFromEngel.Storage_2.CountFinished), ADR(stIo.stIn.aFromEngelRaw[27]), SIZEOF(UINT));
MEMCPY(ADR(stFromEngel.Storage_2.CountEmpty), ADR(stIo.stIn.aFromEngelRaw[29]), SIZEOF(UINT));
END_METHOD

METHOD PRIVATE M_MappingOut : BOOL
VAR_INPUT
END_VAR
MEMCPY(ADR(stIo.stOut.aToEngelRaw[0]), ADR(stToEngel.LifeCounter), SIZEOF(UINT));
MEMCPY(ADR(stIo.stOut.aToEngelRaw[2]), ADR(stToEngel.ErrorID), SIZEOF(UINT));

stIo.stOut.aToEngelRaw[4].0 := stToEngel.Ready;
stIo.stOut.aToEngelRaw[4].1 := stToEngel.Busy;
stIo.stOut.aToEngelRaw[4].2 := False;//stToEngel.Error;
stIo.stOut.aToEngelRaw[4].3 := stToEngel.PermitRoboterHandling;
stIo.stOut.aToEngelRaw[4].4 := stToEngel.PermitStorage_1;
stIo.stOut.aToEngelRaw[4].5 := stToEngel.PermitStorage_2;
stIo.stOut.aToEngelRaw[4].6 := stToEngel.SafetyAreaRequest;
stIo.stOut.aToEngelRaw[4].7 := stToEngel.SafetyDoorRelease;

stIo.stOut.aToEngelRaw[5].0 := stToEngel.JobStatusForStorage_1.CarrierPresent;
stIo.stOut.aToEngelRaw[5].1 := stToEngel.JobStatusForStorage_1.Done;
stIo.stOut.aToEngelRaw[5].2 := stToEngel.JobStatusForStorage_1.Busy;
stIo.stOut.aToEngelRaw[5].3 := stToEngel.JobStatusForStorage_1.Error;
stIo.stOut.aToEngelRaw[5].4 := stToEngel.JobStatusForStorage_2.CarrierPresent;
stIo.stOut.aToEngelRaw[5].5 := stToEngel.JobStatusForStorage_2.Done;
stIo.stOut.aToEngelRaw[5].6 := stToEngel.JobStatusForStorage_2.Busy;
stIo.stOut.aToEngelRaw[5].7 := stToEngel.JobStatusForStorage_2.Error;

//stIo.stOut.aToEngelRaw[6].0 := stToEngel.res.;

MEMCPY(ADR(stIo.stOut.aToEngelRaw[7]), ADR(stToEngel.JobStatusForStorage_1.ErrorID), SIZEOF(UINT));
MEMCPY(ADR(stIo.stOut.aToEngelRaw[9]), ADR(stToEngel.JobStatusForStorage_1.Carrier.CarrierId), SIZEOF(UINT));
MEMCPY(ADR(stIo.stOut.aToEngelRaw[11]), ADR(stToEngel.JobStatusForStorage_1.Carrier.CountMax), SIZEOF(UINT));
MEMCPY(ADR(stIo.stOut.aToEngelRaw[13]), ADR(stToEngel.JobStatusForStorage_1.Carrier.CountUnfinished), SIZEOF(UINT));
MEMCPY(ADR(stIo.stOut.aToEngelRaw[15]), ADR(stToEngel.JobStatusForStorage_1.Carrier.CountFinished), SIZEOF(UINT));
MEMCPY(ADR(stIo.stOut.aToEngelRaw[17]), ADR(stToEngel.JobStatusForStorage_1.Carrier.CountEmpty), SIZEOF(UINT));

MEMCPY(ADR(stIo.stOut.aToEngelRaw[19]), ADR(stToEngel.JobStatusForStorage_2.ErrorID), SIZEOF(UINT));
MEMCPY(ADR(stIo.stOut.aToEngelRaw[21]), ADR(stToEngel.JobStatusForStorage_2.Carrier.CarrierId), SIZEOF(UINT));
MEMCPY(ADR(stIo.stOut.aToEngelRaw[23]), ADR(stToEngel.JobStatusForStorage_2.Carrier.CountMax), SIZEOF(UINT));
MEMCPY(ADR(stIo.stOut.aToEngelRaw[25]), ADR(stToEngel.JobStatusForStorage_2.Carrier.CountUnfinished), SIZEOF(UINT));
MEMCPY(ADR(stIo.stOut.aToEngelRaw[27]), ADR(stToEngel.JobStatusForStorage_2.Carrier.CountFinished), SIZEOF(UINT));
MEMCPY(ADR(stIo.stOut.aToEngelRaw[29]), ADR(stToEngel.JobStatusForStorage_2.Carrier.CountEmpty), SIZEOF(UINT));
END_METHOD

METHOD PROTECTED M_OpModeChanged : BOOL
VAR_INPUT
END_VAR
(*bBusy := FALSE;

IF (eOpMode <> eOpMode_step AND eOpMode <> eOpMode_auto) THEN
	sqAuto.Set(0);
END_IF

fbCamAs.M_Off();
fbCamBs.M_Off();
fbLedAs.M_Off();
fbLedBs.M_Off();*)
END_METHOD

METHOD PUBLIC M_Run : BOOL
VAR_INPUT
END_VAR
// check refs valid
IF NOT __ISVALIDREF(stIO) THEN
	RETURN;
END_IF

M_MappingIn();
M_RUN := SUPER^.M_Run();
stToEngel.LifeCounter := stFromEngel.LifeCounter;
M_MappingOut();

M_DynSettings();
M_DynManual();
M_DynMonitoring();
END_METHOD

METHOD PROTECTED M_Sequence
VAR
END_VAR
// signal mapping (e.g.: enable)
// <- FROM ENGEL
 stSt050IMould.bEnableHG := (NOT (stFromEngel.Moving OR stFromEngel.Error) AND
							stFromEngel.SafetyAreaSafe AND 
							stFromEngel.ParkPosition AND
							stFromEngel.OutsideStorage_1 AND
							stFromEngel.OutsideStorage_2) OR
							bStationDeaktiv; //ToDo: check!!!
							
stSt050IMould.bReqS1Empty := 	stFromEngel.JobForStorage_1.RequestCarrier AND
						   		stFromEngel.JobForStorage_1.Empty;
										 
stSt050IMould.bReqS2Empty := 	stFromEngel.JobForStorage_2.RequestCarrier AND
						   		stFromEngel.JobForStorage_2.Empty;
										 
stSt050IMould.bReqS1Unfinished :=	stFromEngel.JobForStorage_1.RequestCarrier AND
						   			stFromEngel.JobForStorage_1.Unfinished;
										 
stSt050IMould.bReqS2Unfinished :=	stFromEngel.JobForStorage_2.RequestCarrier AND
						   			stFromEngel.JobForStorage_2.Unfinished;
										
stSt050IMould.bReqS1NoCarrier := stFromEngel.JobForStorage_1.RequestNoCarrier;
stSt050IMould.bReqS2NoCarrier := stFromEngel.JobForStorage_2.RequestNoCarrier;

// -> TO ENGEL
stToEngel.PermitRoboterHandling :=
stToEngel.PermitStorage_1 :=
stToEngel.PermitStorage_2 := stSt030IHandling.ActiveCommand.Command = E_St030_Command.eSt030_Command_none;

stToEngel.Busy := stSt030IHandling.ActiveCommand.Command <> E_St030_Command.eSt030_Command_none;
stToEngel.Error := IEvent.ErrorActive;
//ToDo: stToEngel.ErrorID :=

stToEngel.JobStatusForStorage_1.Busy := stSt030IHandling.ActiveCommand.Position = 1 AND
												   (stSt030IHandling.ActiveCommand.Command = E_St030_Command.eSt030_Command_Storage_Get OR 
												   stSt030IHandling.ActiveCommand.Command = E_St030_Command.eSt030_Command_Storage_Put);

											
												   
(*ToDo: IF stSt030IHandling.bCarrierDroppedStorage1 THEN
	stIO.stOut.stToEngel.JobStatusForStorage_1.Carrier.CarrierId := TO_INT(stSt040IStorage.Pallet1.stPallet.ID) ; // ID vom Werkstückträger, Geometrischen Daten werden auf der Engel Steuerung verwaltet
	stIO.stOut.stToEngel.JobStatusForStorage_1.Carrier.CountMax; // maximale Anzahl an Werkstücken die am Werkstückträger abgelegt werden können
	stIO.stOut.stToEngel.JobStatusForStorage_1.Carrier.CountUnfinished; // Anzahl der nicht gegossenen Rohlinge am Werkstückträger
	stIO.stOut.stToEngel.JobStatusForStorage_1.Carrier.CountFinished; // Anzahl der fertigen Werkstücke am Werkstückträger
	stIO.stOut.stToEngel.JobStatusForStorage_1.Carrier.CountEmpty;
	stIO.stOut.stToEngel.JobStatusForStorage_1.CarrierPresent := stSt040IStorage.Pallet1.PalletExists;
	stIO.stOut.stToEngel.JobStatusForStorage_1.Done := TRUE;
ELSIF NOT stSt050IMould.bReqS1Empty AND NOT stSt050IMould.bReqS1Unfinished AND NOT stSt050IMould.bReqS1NoCarrier THEN
	stIO.stOut.stToEngel.JobStatusForStorage_1.Carrier := stFromEngel.Storage_1; // status zurück übernehmen
	stIO.stOut.stToEngel.JobStatusForStorage_1.Done := FALSE;
END_IF *)

(*ToDo: IF stSt030IHandling.bCarrierDroppedStorage1 THEN ...*)

//ToDo: stIO.stOut.stToEngel.SafetyAreaRequest
//ToDo: stIO.stOut.stToEngel.SafetyDoorRelease

// automatic sequence
CASE sqAuto.Step OF
	
	0:	sqAuto.Info.Set("Warte auf Auto Start");
		IF RunCycle AND RunStep THEN
			//sqAuto.Info.Set("Warte auf GRST");
			//IF sqHome.InHome AND bInHome THEN
				sqHome.InHome := FALSE;
				sqAuto.Step := 5;
			//ELSE
			//	StationError.ArgSbAppendWsRaise(stTextlistGlobal.stText_station_not_in_hp);
			//END_IF
		END_IF
		
	5:	IF bStationDeaktiv THEN
			sqAuto.Info.Set("Station deaktiv");
		ELSE
			sqAuto.Step := 10;
		END_IF
		
	10:	sqAuto.Info.Set("Prüfe Startbedingungen");
		//IF NOT stFromEngel.CycleMode THEN
			StationError.ArgSbAppendRaise('Signal Automatikbetrieb Engel fehlt');
		//ELS
		IF stFromEngel.Error THEN
			StationError.ArgSbAppendRaise('Signal Fehler Engel seht an');
		ELSE
			CycleStart();
			bBusy := TRUE;
			sqAuto.Step := 100;
		END_IF

	// work
	100: sqAuto.Info.Set("Automatik");
		IF NOT RunCycle THEN
			stToEngel.Ready := FALSE;
			stToEngel.Busy := FALSE;
			stToEngel.PermitStorage_1 := FALSE;
			stToEngel.PermitStorage_2 := FALSE;
			sqAuto.Step := 900;	
		END_IF
		
	// rdy	
	900: sqAuto.Info.Set("Zyklus beendet");
		CycleEnd();
		sqAuto.Step := 0;

	// error
	1000: sqAuto.Info.Set("Error");
		bStopped := TRUE;
		sqHome.InHome := FALSE;
		bRunHoming := FALSE;

END_CASE
END_METHOD

METHOD INTERNAL M_SetReferences : BOOL
VAR_IN_OUT
	stIoRef : ST_St050_IO;
END_VAR
stIO REF= stIoRef;
M_SetReferences := TRUE;
END_METHOD

METHOD PROTECTED M_Supervision : BOOL
VAR
END_VAR
// chk stopped
IF NOT bRunCycle OR P_Safety.bMachineRequestStop THEN
	IF sqAuto.StepTime > T#20S THEN
		bStopped := TRUE;
	END_IF
END_IF

// Engel SGM
IF stFromEngel.Error THEN
  	ReactToEvent(E_EventReaction.Stop, TcEventSeverity.Error)
		.ArgSbInit('Engel | Error von SGM | ')
	  	.ArgSbAppendAnyRaise(stFromEngel.ErrorID);
END_IF
END_METHOD

/// Reset station logic
{attribute 'object_name' := 'Reset'}
METHOD Reset
VAR
END_VAR
// base logic run
SUPER^.Reset();

// reset objects
//diContinuesNok := 0;

//IF fbCamAs.bError OR NOT RunCycle THEN
	fbCamAs.M_Reset();
	fbCamBs.M_Reset();
	fbLedAs.M_Reset();
	fbLedBs.M_Reset();
//END_IF

//stSt060.bEnable := FALSE;
END_METHOD

END_FUNCTION_BLOCK

// ---- POUs/Components/Device/FB_Device.TcPOU
FUNCTION_BLOCK PUBLIC FB_Device EXTENDS FB_ComponentBase
VAR_INPUT
	// IO reference
	stIn		: ST_DeviceIn;
	//stIO : REFERENCE TO ST_DeviceIO;
END_VAR
VAR_OUTPUT
	bOut		: BOOL;
	fValue		: LREAL;
	stOut		: ST_DeviceOut;
END_VAR
VAR
	// private var's
	bEnable : BOOL;
END_VAR

bOut := stOut.bRun;
fValue := stout.fValue;

PROPERTY PUBLIC Enable : BOOL
GET
Enable := bEnable;
END_GET
SET
bEnable := Enable;
END_SET
END_PROPERTY

METHOD PUBLIC M_Off : BOOL;
VAR_INPUT
END_VAR
stOut.bRun := FALSE;
M_Off := TRUE;
END_METHOD

METHOD PUBLIC M_On : BOOL;
VAR_INPUT
END_VAR
IF bEnable THEN
	stOut.bRun := TRUE;
	M_On := TRUE;
END_IF
END_METHOD

METHOD M_Reset : BOOL
VAR_INPUT
END_VAR
M_Reset := TRUE;
END_METHOD

{attribute 'monitoring' := 'call'}
PROPERTY PUBLIC Value : LREAL
GET
Value := stOut.fValue;
END_GET
SET
stOut.fValue := Value;
END_SET
END_PROPERTY

END_FUNCTION_BLOCK

// ---- POUs/Components/Device/FB_Device_Ui.TcPOU
FUNCTION_BLOCK FB_Device_Ui EXTENDS FB_ManualUiBase
VAR_INPUT
	// enable value input in hmi
	bValueVisible			: BOOL;
	stValueText				: ST_Text;
	
	/// Eingänge zum Bedienen von Visu
	bManualOn				: BOOL;
	bManualOff				: BOOL;
END_VAR
VAR_IN_OUT
	// device reference
	fbDevice		: FB_Device;
	// hmi control IN
	stHMIControlIn	: ST_HMI_MANUAL_DEVICE_IN;
	// hmi control OUT
	stHMIControlOut	: ST_HMI_MANUAL_DEVICE_OUT;		
END_VAR
VAR_OUTPUT
	diColorSelectedItem: UDINT;
	/// 0=Undefiniert
	/// 1=Fehler
	iState: INT;
	diColorState	: UDINT;
	sState			: STRING;
	stState			: ST_Text;	
	/// 0=Off; 
	/// 1=On; 
	/// 2=Undefiniert... 

	///Darstellung der Controls für das Object 
	///0=Unsichtbar
	///1=Sichtbar Unselektiert
	///2=Sichtbar Selektiert	
END_VAR

stName := fbDevice.stName;

IF (diSelectedObjectIndex = diObjectIndex) AND bEnableManual THEN
	bManualActive := TRUE;
	stHMIControlOut.bVisible := TRUE;
	stHMIControlOut.stObjectName := fbDevice.stName;
	stHMIControlOut.bValueVisible := bValueVisible;
	stHMIControlOut.stValueText := stValueText;
	stHMIControlOut.stButtonOn.stName := CONST.stTextListGlobal.stText_On;
	stHMIControlOut.stButtonOff.stName := CONST.stTextListGlobal.stText_Off;

	IF stHMIControlIn.stButtonOn.bClick THEN
		fbDevice.M_On();
	ELSIF stHMIControlIn.stButtonOff.bClick THEN
		fbDevice.M_Off();
	END_IF
	fbDevice.Value := stHMIControlIn.fValue;

	stHMIControlOut.stButtonOn.stColor.color := F_ColorToStringHexColor(STATICS.stColor.Theme);
	stHMIControlOut.stButtonOff.stColor.color := F_ColorToStringHexColor(STATICS.stColor.Red);
	IF fbDevice.stOut.bRun THEN
		stHMIControlOut.stButtonOn.stColor.color := F_ColorToStringHexColor(STATICS.stColor.LimeGreen);
	END_IF
	
	stHMIControlOut.stState	:= 	stState;
ELSIF bManualActive THEN
	bManualActive := FALSE;
	stHMIControlOut.bVisible := FALSE;
END_IF

IF bManualOn THEN
	fbDevice.M_On();
END_IF

IF bManualOff THEN
	fbDevice.M_Off();
END_IF

IF fbDevice.stOut.bRun THEN
	stState := stTextListGlobal.stText_On;
ELSE
	stState := stTextListGlobal.stText_Off;	
END_IF

A_StateMapping();

ACTION A_StateMapping:
IF NOT __ISVALIDREF(stStateObject) THEN
	RETURN;
END_IF

// state mapping
stStateObject.stState := stState;
stStateObject.nIndexColor := diColorSelectedItem;
END_ACTION

END_FUNCTION_BLOCK

// ---- POUs/Components/AxisDriver/FB_AxisCoupleSync2.TcPOU
FUNCTION_BLOCK FB_AxisCoupleSync2
VAR_IN_OUT
	fbAxis_Master			: FB_AxisDriver;
	stAxisMasterREF			: AXIS_REF;
	fbAxis_Slave			: FB_AxisDriver;	
END_VAR
VAR_INPUT
	eAxisMaster					:E_Axis;
	
	eOpModeStation				:E_OpMode;
	/// Koppeln
	bCoupleOn					:BOOL;
	/// Achsen synchronisieren
	bSyncOn						:BOOL;
	/// Tipppen
	bJog						:BOOL;;
	/// Sync Geschwindigkeit
	fVelocity					:REAL := 1;
	
	/// Endschalter Master (Oeffner)
	bRefSwitchMaster			:BOOL;
	/// Endschalter Slave (Oeffner)
	bRefSwitchSlave				:BOOL;
END_VAR
VAR_OUTPUT
	bCoupled				:BOOL;
	bCoupleStateOK			:BOOL;
	bSyncActiv				:BOOL;
	bSyncDone				:BOOL;
	bSyncError				:BOOL;
END_VAR
VAR
	iStepSync	:INT;
	
	iStepKoppeln		:INT;
	negSync			:F_TRIG;
	tonTimeOutGear	:TON;
END_VAR

(*
	Baustein um 2 Achsen zu koppeln und 
	auf Ref. Schalter zu Synchronisieren
*)
// Timer, Flanken
tonTimeOutGear(PT := T#2S);


negSync(CLK := bSyncOn);
IF negSync.Q THEN
	IF fbAxis_Master.Moving THEN
		fbAxis_Master.Halt();
	END_IF
	IF fbAxis_Slave.Moving THEN
		fbAxis_Slave.Halt();
	END_IF
END_IF

IF NOT bSyncOn OR eOpModeStation <> E_OpMode.eOpMode_Manual THEN
	iStepSync := 0;
	bSyncActiv := FALSE;
	bSyncDone := FALSE;
	A_Couple();
	RETURN;
END_IF

iStepKoppeln := 0;
bCoupled := FALSE;


CASE iStepSync OF
	
	0:
		bSyncError := FALSE;
		bSyncDone := FALSE;
		bSyncActiv := TRUE;
		iStepSync := 10;
		
		// Einkoppeln
	10:
		fbAxis_Slave.GearIn(1, eAxisMaster, stAxisMasterREF);
		tonTimeOutGear(IN := FALSE);
		iStepSync := 20;
		
	20:
		tonTimeOutGear(IN := TRUE);
		IF fbAxis_Slave.Coupled AND
		NOT fbAxis_Slave.bError THEN
			iStepSync := 30;
		ELSIF fbAxis_Slave.bError THEN
			iStepSync := 800; // Fehler
		ELSIF tonTimeOutGear.Q THEN
			tonTimeOutGear(IN := FALSE);
			iStepSync := 0;
		END_IF		
		
		
		// Master negative Richtung tippen bis Endschalter
	30:
		iStepSync := 50;
(*		fbAxis_Master.JogExVel((bJog AND bFreigabe_N AND bRefSwitchMaster AND bRefSwitchSlave), 
								FALSE, fVelocity, E_JogMode.MC_JOGMODE_CONTINOUS);
		IF NOT bRefSwitchMaster OR NOT bRefSwitchSlave THEN
			fbAxis_Master.Halt();
			iStepSync := 50;
		ELSIF fbAxis_Master.Error OR fbAxis_Slave.Error THEN
			iStepSync := 800;
		END_IF
*)
		
	50:
		IF NOT fbAxis_Master.Moving THEN
			iStepSync := 60;			
		ELSE
			fbAxis_Master.Halt();
		END_IF
		
		// Auskuppeln
	60:
		fbAxis_Slave.GearOut();
		tonTimeOutGear(IN := FALSE);
		iStepSync := 65;
		
	65:
		tonTimeOutGear(IN := TRUE);
		IF NOT fbAxis_Slave.Coupled THEN
			IF fbAxis_Slave.Moving THEN
				fbAxis_Slave.Halt();
			END_IF
			iStepSync := 100;
			
		ELSIF tonTimeOutGear.Q THEN
			tonTimeOutGear(IN := FALSE);
			iStepSync := 60;
		END_IF		
	
		
		// mit Slave auf MasterPos fahren
	100:
		IF F_TargetWindowReachedAxisRef(fbAxis_Slave,
										fbAxis_Master.Position, 0.01) AND
		NOT fbAxis_Slave.Moving THEN
			iStepSync := 110;
			
		ELSIF bJog THEN
			IF NOT fbAxis_Slave.Moving THEN
				fbAxis_Slave.MoveAbsExVel(fbAxis_Master.Position, fVelocity);
			END_IF
		
		ELSIF fbAxis_Slave.Moving THEN
			fbAxis_Slave.Halt();

		ELSIF fbAxis_Master.bError OR fbAxis_Slave.bError THEN
			iStepSync := 800;
		END_IF
		
	110:
		iStepSync := 200;
		
		
		// Einkoppeln
	200:
		fbAxis_Slave.GearIn(1, eAxisMaster, stAxisMasterREF);
		tonTimeOutGear(IN := FALSE);
		iStepSync := 210;
		
	210:
		tonTimeOutGear(IN := TRUE);
		IF fbAxis_Slave.Coupled AND
		NOT fbAxis_Slave.bError THEN
			iStepSync := 500;
		ELSIF fbAxis_Slave.bError THEN
			iStepSync := 800; // Fehler
		ELSIF tonTimeOutGear.Q THEN
			tonTimeOutGear(IN := FALSE);
			iStepSync := 0;
		END_IF			
		
		
		// FERTIG
	500:
		bSyncActiv := FALSE;
		bSyncDone := TRUE;
		
		
// Fehler
	800:
		bSyncError := TRUE;
		IF fbAxis_Master.Moving THEN
			fbAxis_Master.Halt();
		END_IF
		IF fbAxis_Slave.Moving THEN
			fbAxis_Slave.Halt();
		END_IF		
		iStepSync := 810;	
	
	810:
		bSyncError := TRUE;
		IF NOT fbAxis_Master.bError AND
		NOT fbAxis_Slave.bError THEN
			iStepSync := 0;		
		END_IF
		
END_CASE

ACTION A_Couple:
// Antriebe Transfer koppeln
CASE iStepKoppeln OF
	
	0:
		IF bCoupleOn THEN
			bCoupleStateOK := FALSE;
			iStepKoppeln := 100; // Gear In
		ELSE					
			bCoupleStateOK := FALSE;
			iStepKoppeln := 500; // Gear Out
		END_IF
	

// Koppeln

		// kein Fehler
	100:
		IF NOT fbAxis_Master.bError AND
		fbAxis_Master.Operational AND
		NOT fbAxis_Slave.bError AND
		fbAxis_Slave.Operational THEN
			iStepKoppeln := 110;
		ELSIF NOT bCoupleOn THEN
			iStepKoppeln := 0;
		ELSE
			iStepKoppeln := 800; // Fehler
		END_IF
		
		// koppeln
	110:
		fbAxis_Slave.GearIn(1, eAxisMaster, stAxisMasterREF);
		tonTimeOutGear(IN := FALSE);
		iStepKoppeln := 120;
		
	120:
		tonTimeOutGear(IN := TRUE);
		IF fbAxis_Slave.Coupled AND
		NOT fbAxis_Slave.bError THEN
			iStepKoppeln := 130;
		ELSIF fbAxis_Slave.bError THEN
			iStepKoppeln := 800; // Fehler
		ELSIF tonTimeOutGear.Q THEN
			tonTimeOutGear(IN := FALSE);
			iStepKoppeln := 0;
		ELSIF NOT bCoupleOn THEN
			iStepKoppeln := 0;
		END_IF
	
		// Ueberwache Kopplung
	130:
		tonTimeOutGear(IN := FALSE);
		bCoupleStateOK := TRUE;
		// Koppeln aus
		IF NOT bCoupleOn THEN
			iStepKoppeln := 0;
		END_IF
		// Slave Antrieb hat Fehler und Master fährt -> Stopp Master
		IF fbAxis_Slave.bError AND fbAxis_Master.Moving THEN
			fbAxis_Master.Halt();
		END_IF
		// Master Antrieb hat Fehler -> für Kopplung egal
		IF fbAxis_Master.bError THEN
			;
		END_IF
		
		// Slave nicht mehr gekoppelt --> neu koppeln
		IF NOT fbAxis_Slave.Coupled THEN
			IF fbAxis_Master.Moving THEN
				fbAxis_Master.Halt();				
			END_IF
			iStepKoppeln := 0;
		END_IF
	

// Entkoppeln

		// Stoppen
	500:
		IF fbAxis_Master.Moving THEN
			fbAxis_Master.Halt();				
		ELSE
			iStepKoppeln := 510;
		END_IF

	510:
		fbAxis_Slave.GearOut();
		tonTimeOutGear(IN := FALSE);
		iStepKoppeln := 520;
		
	520:
		tonTimeOutGear(IN := TRUE);
		IF NOT fbAxis_Slave.Coupled THEN
			IF fbAxis_Slave.Moving THEN
				fbAxis_Slave.Halt();
			END_IF
			iStepKoppeln := 530;
		ELSIF tonTimeOutGear.Q THEN
			tonTimeOutGear(IN := FALSE);
			iStepKoppeln := 0;
		END_IF

		// Achse soll wieder koppeln
	530:
		bCoupleStateOK := TRUE;
		IF bCoupleOn THEN
			iStepKoppeln := 0;
		END_IF
		// Status darf sich nicht ändern -> neu einstellen
		IF fbAxis_Slave.Coupled THEN
			iStepKoppeln := 0;
		END_IF
		
		
// Fehler
	800:
		bCoupleStateOK := FALSE;
		IF NOT fbAxis_Master.bError AND
		NOT fbAxis_Slave.bError THEN
			iStepKoppeln := 0;		
		END_IF
		
END_CASE

bCoupled := bCoupleStateOK AND fbAxis_Slave.Coupled;
END_ACTION

END_FUNCTION_BLOCK

// ---- POUs/Components/AxisDriver/Utilities/F_TargetWindowReachedAxisRef.TcPOU
FUNCTION F_TargetWindowReachedAxisRef : BOOL
VAR_IN_OUT
	/// Achse als Referenz
	fbAxis		:FB_AxisDriver;
END_VAR
VAR_INPUT
	fTargetPos: LREAL;
	fWindow: LREAL;
END_VAR


F_TargetWindowReachedAxisRef := fbAxis.Position >= (fTargetPos - fWindow) AND fbAxis.Position <= (fTargetPos + fWindow);

END_FUNCTION

